(* IEC 61131-3 sources: cc_kush_rewrite/POUs (part 2) *)

// DO MODULES MAPPING (350-399)

// Модуль DO1 (350-351): Бункеры 1-2 - Управление ЧРП
FC_ModbusWriteBool(pRegisters := ADR(awModbusInputRegisters), iRegisterIndex := 350, iBitIndex := 0, xValue := stBunker[1].MotorVibFeeder[1].VFD.qxStart);
FC_ModbusWriteBool(pRegisters := ADR(awModbusInputRegisters), iRegisterIndex := 350, iBitIndex := 1, xValue := stBunker[1].MotorVibFeeder[1].VFD.qxResetFailure);
FC_ModbusWriteBool(pRegisters := ADR(awModbusInputRegisters), iRegisterIndex := 350, iBitIndex := 2, xValue := stBunker[1].MotorVibFeeder[2].VFD.qxStart);
FC_ModbusWriteBool(pRegisters := ADR(awModbusInputRegisters), iRegisterIndex := 350, iBitIndex := 3, xValue := stBunker[1].MotorVibFeeder[2].VFD.qxResetFailure);
FC_ModbusWriteBool(pRegisters := ADR(awModbusInputRegisters), iRegisterIndex := 350, iBitIndex := 4, xValue := stBunker[1].MotorVibrator[1].VFD.qxStart);
FC_ModbusWriteBool(pRegisters := ADR(awModbusInputRegisters), iRegisterIndex := 350, iBitIndex := 5, xValue := stBunker[1].MotorVibrator[1].VFD.qxResetFailure);
FC_ModbusWriteBool(pRegisters := ADR(awModbusInputRegisters), iRegisterIndex := 350, iBitIndex := 6, xValue := stBunker[1].MotorVibrator[2].VFD.qxStart);
FC_ModbusWriteBool(pRegisters := ADR(awModbusInputRegisters), iRegisterIndex := 350, iBitIndex := 7, xValue := stBunker[1].MotorVibrator[2].VFD.qxResetFailure);
FC_ModbusWriteBool(pRegisters := ADR(awModbusInputRegisters), iRegisterIndex := 350, iBitIndex := 8, xValue := stBunker[1].MotorVibrator[3].VFD.qxStart);
FC_ModbusWriteBool(pRegisters := ADR(awModbusInputRegisters), iRegisterIndex := 350, iBitIndex := 9, xValue := stBunker[1].MotorVibrator[3].VFD.qxResetFailure);
FC_ModbusWriteBool(pRegisters := ADR(awModbusInputRegisters), iRegisterIndex := 350, iBitIndex := 10, xValue := stBunker[1].MotorVibrator[4].VFD.qxStart);
FC_ModbusWriteBool(pRegisters := ADR(awModbusInputRegisters), iRegisterIndex := 350, iBitIndex := 11, xValue := stBunker[1].MotorVibrator[4].VFD.qxResetFailure);
FC_ModbusWriteBool(pRegisters := ADR(awModbusInputRegisters), iRegisterIndex := 350, iBitIndex := 12, xValue := stBunker[2].MotorVibFeeder[1].VFD.qxStart);
FC_ModbusWriteBool(pRegisters := ADR(awModbusInputRegisters), iRegisterIndex := 350, iBitIndex := 13, xValue := stBunker[2].MotorVibFeeder[1].VFD.qxResetFailure);
FC_ModbusWriteBool(pRegisters := ADR(awModbusInputRegisters), iRegisterIndex := 350, iBitIndex := 14, xValue := stBunker[2].MotorVibFeeder[2].VFD.qxStart);
FC_ModbusWriteBool(pRegisters := ADR(awModbusInputRegisters), iRegisterIndex := 350, iBitIndex := 15, xValue := stBunker[2].MotorVibFeeder[2].VFD.qxResetFailure);

FC_ModbusWriteBool(pRegisters := ADR(awModbusInputRegisters), iRegisterIndex := 351, iBitIndex := 0, xValue := stBunker[2].MotorVibrator[1].VFD.qxStart);
FC_ModbusWriteBool(pRegisters := ADR(awModbusInputRegisters), iRegisterIndex := 351, iBitIndex := 1, xValue := stBunker[2].MotorVibrator[1].VFD.qxResetFailure);
FC_ModbusWriteBool(pRegisters := ADR(awModbusInputRegisters), iRegisterIndex := 351, iBitIndex := 2, xValue := stBunker[2].MotorVibrator[2].VFD.qxStart);
FC_ModbusWriteBool(pRegisters := ADR(awModbusInputRegisters), iRegisterIndex := 351, iBitIndex := 3, xValue := stBunker[2].MotorVibrator[2].VFD.qxResetFailure);
FC_ModbusWriteBool(pRegisters := ADR(awModbusInputRegisters), iRegisterIndex := 351, iBitIndex := 4, xValue := stBunker[2].MotorVibrator[3].VFD.qxStart);
FC_ModbusWriteBool(pRegisters := ADR(awModbusInputRegisters), iRegisterIndex := 351, iBitIndex := 5, xValue := stBunker[2].MotorVibrator[3].VFD.qxResetFailure);
FC_ModbusWriteBool(pRegisters := ADR(awModbusInputRegisters), iRegisterIndex := 351, iBitIndex := 6, xValue := stBunker[2].MotorVibrator[4].VFD.qxStart);
FC_ModbusWriteBool(pRegisters := ADR(awModbusInputRegisters), iRegisterIndex := 351, iBitIndex := 7, xValue := stBunker[2].MotorVibrator[4].VFD.qxResetFailure);

// Модуль DO2 (352-353): Бункер 3, Конвейер, Отвалообразователь - Управление ЧРП
FC_ModbusWriteBool(pRegisters := ADR(awModbusInputRegisters), iRegisterIndex := 352, iBitIndex := 0, xValue := stBunker[3].MotorVibFeeder[1].VFD.qxStart);
FC_ModbusWriteBool(pRegisters := ADR(awModbusInputRegisters), iRegisterIndex := 352, iBitIndex := 1, xValue := stBunker[3].MotorVibFeeder[1].VFD.qxResetFailure);
FC_ModbusWriteBool(pRegisters := ADR(awModbusInputRegisters), iRegisterIndex := 352, iBitIndex := 2, xValue := stBunker[3].MotorVibFeeder[2].VFD.qxStart);
FC_ModbusWriteBool(pRegisters := ADR(awModbusInputRegisters), iRegisterIndex := 352, iBitIndex := 3, xValue := stBunker[3].MotorVibFeeder[2].VFD.qxResetFailure);
FC_ModbusWriteBool(pRegisters := ADR(awModbusInputRegisters), iRegisterIndex := 352, iBitIndex := 4, xValue := stBunker[3].MotorVibrator[1].VFD.qxStart);
FC_ModbusWriteBool(pRegisters := ADR(awModbusInputRegisters), iRegisterIndex := 352, iBitIndex := 5, xValue := stBunker[3].MotorVibrator[1].VFD.qxResetFailure);
FC_ModbusWriteBool(pRegisters := ADR(awModbusInputRegisters), iRegisterIndex := 352, iBitIndex := 6, xValue := stBunker[3].MotorVibrator[2].VFD.qxStart);
FC_ModbusWriteBool(pRegisters := ADR(awModbusInputRegisters), iRegisterIndex := 352, iBitIndex := 7, xValue := stBunker[3].MotorVibrator[2].VFD.qxResetFailure);
FC_ModbusWriteBool(pRegisters := ADR(awModbusInputRegisters), iRegisterIndex := 352, iBitIndex := 8, xValue := stBunker[3].MotorVibrator[3].VFD.qxStart);
FC_ModbusWriteBool(pRegisters := ADR(awModbusInputRegisters), iRegisterIndex := 352, iBitIndex := 9, xValue := stBunker[3].MotorVibrator[3].VFD.qxResetFailure);
FC_ModbusWriteBool(pRegisters := ADR(awModbusInputRegisters), iRegisterIndex := 352, iBitIndex := 10, xValue := stBunker[3].MotorVibrator[4].VFD.qxStart);
FC_ModbusWriteBool(pRegisters := ADR(awModbusInputRegisters), iRegisterIndex := 352, iBitIndex := 11, xValue := stBunker[3].MotorVibrator[4].VFD.qxResetFailure);
FC_ModbusWriteBool(pRegisters := ADR(awModbusInputRegisters), iRegisterIndex := 352, iBitIndex := 12, xValue := stConveyor.MotorConveyor[1].VFD.qxStart);
FC_ModbusWriteBool(pRegisters := ADR(awModbusInputRegisters), iRegisterIndex := 352, iBitIndex := 13, xValue := stConveyor.MotorConveyor[1].VFD.qxResetFailure);
FC_ModbusWriteBool(pRegisters := ADR(awModbusInputRegisters), iRegisterIndex := 352, iBitIndex := 14, xValue := stConveyor.MotorConveyor[2].VFD.qxStart);
FC_ModbusWriteBool(pRegisters := ADR(awModbusInputRegisters), iRegisterIndex := 352, iBitIndex := 15, xValue := stConveyor.MotorConveyor[2].VFD.qxResetFailure);

FC_ModbusWriteBool(pRegisters := ADR(awModbusInputRegisters), iRegisterIndex := 353, iBitIndex := 0, xValue := stDumper.MotorConveyor[1].VFD.qxStart);
FC_ModbusWriteBool(pRegisters := ADR(awModbusInputRegisters), iRegisterIndex := 353, iBitIndex := 1, xValue := stDumper.MotorConveyor[1].VFD.qxResetFailure);
FC_ModbusWriteBool(pRegisters := ADR(awModbusInputRegisters), iRegisterIndex := 353, iBitIndex := 2, xValue := stDumper.MotorConveyor[2].VFD.qxStart);
FC_ModbusWriteBool(pRegisters := ADR(awModbusInputRegisters), iRegisterIndex := 353, iBitIndex := 3, xValue := stDumper.MotorConveyor[2].VFD.qxResetFailure);
FC_ModbusWriteBool(pRegisters := ADR(awModbusInputRegisters), iRegisterIndex := 353, iBitIndex := 4, xValue := stDumper.MotorRotation[1].VFD.qxStart);
FC_ModbusWriteBool(pRegisters := ADR(awModbusInputRegisters), iRegisterIndex := 353, iBitIndex := 5, xValue := stDumper.MotorRotation[1].qxVFDReverseStart);
FC_ModbusWriteBool(pRegisters := ADR(awModbusInputRegisters), iRegisterIndex := 353, iBitIndex := 6, xValue := stDumper.MotorRotation[1].VFD.qxResetFailure);
FC_ModbusWriteBool(pRegisters := ADR(awModbusInputRegisters), iRegisterIndex := 353, iBitIndex := 7, xValue := stDumper.MotorRotation[2].VFD.qxStart);
FC_ModbusWriteBool(pRegisters := ADR(awModbusInputRegisters), iRegisterIndex := 353, iBitIndex := 8, xValue := stDumper.MotorRotation[2].qxVFDReverseStart);
FC_ModbusWriteBool(pRegisters := ADR(awModbusInputRegisters), iRegisterIndex := 353, iBitIndex := 9, xValue := stDumper.MotorRotation[2].VFD.qxResetFailure);

// Модуль DO3 (354-355): Контакторы и общие выходы
FC_ModbusWriteBool(pRegisters := ADR(awModbusInputRegisters), iRegisterIndex := 354, iBitIndex := 0, xValue := stConveyor.MotorConveyor[1].qxKM_Power);
FC_ModbusWriteBool(pRegisters := ADR(awModbusInputRegisters), iRegisterIndex := 354, iBitIndex := 1, xValue := stConveyor.MotorConveyor[2].qxKM_Power);
FC_ModbusWriteBool(pRegisters := ADR(awModbusInputRegisters), iRegisterIndex := 354, iBitIndex := 2, xValue := stDumper.MotorConveyor[1].qxKM_Power);
FC_ModbusWriteBool(pRegisters := ADR(awModbusInputRegisters), iRegisterIndex := 354, iBitIndex := 3, xValue := stDumper.MotorConveyor[2].qxKM_Power);
FC_ModbusWriteBool(pRegisters := ADR(awModbusInputRegisters), iRegisterIndex := 354, iBitIndex := 4, xValue := stDumper.MotorRotation[1].qxKM_Power);
FC_ModbusWriteBool(pRegisters := ADR(awModbusInputRegisters), iRegisterIndex := 354, iBitIndex := 5, xValue := stDumper.MotorRotation[2].qxKM_Power);
FC_ModbusWriteBool(pRegisters := ADR(awModbusInputRegisters), iRegisterIndex := 354, iBitIndex := 6, xValue := stBunker[1].MotorVibFeeder[1].qxKM_Power);
FC_ModbusWriteBool(pRegisters := ADR(awModbusInputRegisters), iRegisterIndex := 354, iBitIndex := 7, xValue := stBunker[1].MotorVibFeeder[2].qxKM_Power);
FC_ModbusWriteBool(pRegisters := ADR(awModbusInputRegisters), iRegisterIndex := 354, iBitIndex := 8, xValue := stBunker[1].MotorVibrator[1].qxKM_Power);
FC_ModbusWriteBool(pRegisters := ADR(awModbusInputRegisters), iRegisterIndex := 354, iBitIndex := 9, xValue := stBunker[1].MotorVibrator[2].qxKM_Power);
FC_ModbusWriteBool(pRegisters := ADR(awModbusInputRegisters), iRegisterIndex := 354, iBitIndex := 10, xValue := stBunker[1].MotorVibrator[3].qxKM_Power);
FC_ModbusWriteBool(pRegisters := ADR(awModbusInputRegisters), iRegisterIndex := 354, iBitIndex := 11, xValue := stBunker[1].MotorVibrator[4].qxKM_Power);
FC_ModbusWriteBool(pRegisters := ADR(awModbusInputRegisters), iRegisterIndex := 354, iBitIndex := 12, xValue := stBunker[2].MotorVibFeeder[1].qxKM_Power);
FC_ModbusWriteBool(pRegisters := ADR(awModbusInputRegisters), iRegisterIndex := 354, iBitIndex := 13, xValue := stBunker[2].MotorVibFeeder[2].qxKM_Power);
FC_ModbusWriteBool(pRegisters := ADR(awModbusInputRegisters), iRegisterIndex := 354, iBitIndex := 14, xValue := stBunker[2].MotorVibrator[1].qxKM_Power);
FC_ModbusWriteBool(pRegisters := ADR(awModbusInputRegisters), iRegisterIndex := 354, iBitIndex := 15, xValue := stBunker[2].MotorVibrator[2].qxKM_Power);

FC_ModbusWriteBool(pRegisters := ADR(awModbusInputRegisters), iRegisterIndex := 355, iBitIndex := 0, xValue := stBunker[2].MotorVibrator[3].qxKM_Power);
FC_ModbusWriteBool(pRegisters := ADR(awModbusInputRegisters), iRegisterIndex := 355, iBitIndex := 1, xValue := stBunker[2].MotorVibrator[4].qxKM_Power);
FC_ModbusWriteBool(pRegisters := ADR(awModbusInputRegisters), iRegisterIndex := 355, iBitIndex := 2, xValue := stBunker[3].MotorVibFeeder[1].qxKM_Power);
FC_ModbusWriteBool(pRegisters := ADR(awModbusInputRegisters), iRegisterIndex := 355, iBitIndex := 3, xValue := stBunker[3].MotorVibFeeder[2].qxKM_Power);
FC_ModbusWriteBool(pRegisters := ADR(awModbusInputRegisters), iRegisterIndex := 355, iBitIndex := 4, xValue := stBunker[3].MotorVibrator[1].qxKM_Power);
FC_ModbusWriteBool(pRegisters := ADR(awModbusInputRegisters), iRegisterIndex := 355, iBitIndex := 5, xValue := stBunker[3].MotorVibrator[2].qxKM_Power);
FC_ModbusWriteBool(pRegisters := ADR(awModbusInputRegisters), iRegisterIndex := 355, iBitIndex := 6, xValue := stBunker[3].MotorVibrator[3].qxKM_Power);
FC_ModbusWriteBool(pRegisters := ADR(awModbusInputRegisters), iRegisterIndex := 355, iBitIndex := 7, xValue := stBunker[3].MotorVibrator[4].qxKM_Power);
FC_ModbusWriteBool(pRegisters := ADR(awModbusInputRegisters), iRegisterIndex := 355, iBitIndex := 8, xValue := stConveyor.xHLA);
FC_ModbusWriteBool(pRegisters := ADR(awModbusInputRegisters), iRegisterIndex := 355, iBitIndex := 10, xValue := stDumper.xHLA);
FC_ModbusWriteBool(pRegisters := ADR(awModbusInputRegisters), iRegisterIndex := 355, iBitIndex := 11, xValue := stCommonSignals.qx6KM1);
FC_ModbusWriteBool(pRegisters := ADR(awModbusInputRegisters), iRegisterIndex := 355, iBitIndex := 12, xValue := stConveyor.qxBreakerConveyor);
FC_ModbusWriteBool(pRegisters := ADR(awModbusInputRegisters), iRegisterIndex := 355, iBitIndex := 13, xValue := stDumper.qxBreakerConveyor);
FC_ModbusWriteBool(pRegisters := ADR(awModbusInputRegisters), iRegisterIndex := 355, iBitIndex := 14, xValue := stDumper.qxBreakerRotation);

// Модуль DO4 (356-357): Светофоры бункеров
FC_ModbusWriteBool(pRegisters := ADR(awModbusInputRegisters), iRegisterIndex := 356, iBitIndex := 0, xValue := stBunker[1].qxLightRed);
FC_ModbusWriteBool(pRegisters := ADR(awModbusInputRegisters), iRegisterIndex := 356, iBitIndex := 1, xValue := stBunker[1].qxLightYellow);
FC_ModbusWriteBool(pRegisters := ADR(awModbusInputRegisters), iRegisterIndex := 356, iBitIndex := 2, xValue := stBunker[1].qxLightGreen);
FC_ModbusWriteBool(pRegisters := ADR(awModbusInputRegisters), iRegisterIndex := 356, iBitIndex := 3, xValue := stBunker[2].qxLightRed);
FC_ModbusWriteBool(pRegisters := ADR(awModbusInputRegisters), iRegisterIndex := 356, iBitIndex := 4, xValue := stBunker[2].qxLightYellow);
FC_ModbusWriteBool(pRegisters := ADR(awModbusInputRegisters), iRegisterIndex := 356, iBitIndex := 5, xValue := stBunker[2].qxLightGreen);
FC_ModbusWriteBool(pRegisters := ADR(awModbusInputRegisters), iRegisterIndex := 356, iBitIndex := 6, xValue := stBunker[3].qxLightRed);
FC_ModbusWriteBool(pRegisters := ADR(awModbusInputRegisters), iRegisterIndex := 356, iBitIndex := 7, xValue := stBunker[3].qxLightYellow);
FC_ModbusWriteBool(pRegisters := ADR(awModbusInputRegisters), iRegisterIndex := 356, iBitIndex := 8, xValue := stBunker[3].qxLightGreen);

END_FUNCTION

(* ---- FB_BunkerControl.st ---- *)
FUNCTION_BLOCK FB_BunkerControl
VAR_INPUT
	Bunker : REFERENCE TO ST_Bunker;
	xLocalMode : BOOL; // TRUE = местный режим (ПМУ), FALSE = дистанционный режим (SCADA)
	xStart : BOOL; // Команда запуска вибропитателей (дистанционный режим)
	xStop : BOOL; // Команда остановки (дистанционный режим)
	xEmergencyStopVibFeeder : BOOL; // Аварийная остановка вибропитателей (переводит бункер в ERROR)
	xEmergencyStopVibrator : BOOL; // Аварийная остановка вибраторов (только отключает вибраторы)
	xReset : BOOL; // Сброс ошибок
	irManualFrequency : REAL; // Частота вибропитателей для ручного режима управления
	irManualFrequencyVibrator : REAL; // Частота вибраторов для ручного режима управления
END_VAR
VAR_OUTPUT
	eStage : E_StageWithPreStartAlarm; // Текущая стадия запуска вибропитателей
	eStageToSCADA : E_ScadaStatesDevice; // Передача состояния скаде
END_VAR
VAR
	i : INT;
	_rtStartCmd, _rtStopCmd : R_TRIG; // Детекторы фронтов для команд

	// Локальные переменные для управления в режиме МЕСТНЫЙ
	_rtStartKM, _rtStopKM : R_TRIG;
	_rtStartVFD, _rtStopVFD : R_TRIG;

	// Объединенные команды (ПМУ или SCADA в зависимости от режима)
	xStartCommand : BOOL; // Фактическая команда запуска (из ПМУ или SCADA)
	xStopCommand : BOOL; // Фактическая команда остановки (из ПМУ или SCADA)

	// ФБ управления
	fbPneumoControl : FB_PneumoCollapseControl;

	// Таймеры для автоматического цикла вибраторов
	tonVibratorActive : TON;  // Таймер активной работы вибраторов
	tonVibratorPause : TON;   // Таймер паузы вибраторов

	// Автомат состояний для запуска вибропитателей
	STAGE : E_StageWithPreStartAlarm := E_StageWithPreStartAlarm.IDLE;

	// Состояние схемы контакторов (TRUE = схема собрана, FALSE = схема разобрана)
	xCircuitBuilt : BOOL := FALSE;
	xCircuitBuiltVibrator : BOOL := FALSE;

	// Целевые частоты для моторов вибропитателей
	rTargetFreqVibFeeder1 : REAL := 0.0;
	rTargetFreqVibFeeder2 : REAL := 0.0;

	// Флаг активного запуска вибраторов в ручном режиме
	xVibratorManualRunActive : BOOL := FALSE;

	// Флаг текущей активности вибраторов в автоматическом режиме
	xVibratorAutoActive : BOOL := FALSE;

	// Таймеры контроля выполнения команд
	fbTimerStarting : TON; // Тайм-аут запуска (STARTING → WORK)
	fbTimerStopping : TON; // Тайм-аут остановки (WORK → IDLE)

END_VAR

// ========================================
// FB_BunkerControl - Управление бункером
// ========================================
//
// РЕЖИМЫ УПРАВЛЕНИЯ:
//
// 1. МЕСТНЫЙ РЕЖИМ (xLocalMode = TRUE):
//    - Команды берутся с кнопок ПМУ (Bunker.fbBtnStart, fbBtnStop)
//    - ПУСК/СТОП вибропитателей по фронтам кнопок
//    - Автоматически устанавливает eStateRemote = Manual
//
// 2. ДИСТАНЦИОННЫЙ РЕЖИМ (xLocalMode = FALSE):
//    - Команды берутся из входов ФБ (xStart, xStop)
//    - Режим устанавливается через SCADA (Manual/Remote/Auto)
//
// УПРАВЛЕНИЕ ВИБРОПИТАТЕЛЯМИ:
// - ПУСК: включение вибропитателей с заданной частотой
// - СТОП: остановка вибропитателей
// - Частота: Auto - от ПИД, Manual/Repair - от irManualFrequency
//
// УПРАВЛЕНИЕ ВИБРАТОРАМИ:
// - Независимо от режима вибропитателей
// - Режимы:
//   * Auto - циклическая работа по таймеру (ACTIVE ↔ PAUSE)
//     - Работает только в стадии WORK вибропитателей
//     - Параметры: VIBRATOR_SETTINGS.TIME_ACTIVE, TIME_PAUSE_VIBRATOR
//     - Частота: irManualFrequencyVibrator
//   * Manual - выборочное управление через cmdAddVib1..4
//     - СТАРТ/СТОП по командам cmdStartVibrator/cmdStopVibrator
//     - Частота: irManualFrequencyVibrator
//   * Repair - все вибраторы остановлены
//
// ========================================

// ========================================
// ИНИЦИАЛИЗАЦИЯ СИГНАЛОВ С ФИЛЬТРАЦИЕЙ ДРЕБЕЗГА
// ========================================

// Положение люка - с фильтрацией дребезга
Bunker.fbStateHatch(
	ixSignal := , // Подключить физический вход
	xEnableRattlingFilter := TRUE,
	tStabilityTime := T#100MS
);

// ПМУ - СТАРТ - с фильтрацией дребезга
Bunker.fbBtnStart(
	ixSignal := , // Подключить физический вход
	xEnableRattlingFilter := TRUE,
	tStabilityTime := T#100MS
);

// ПМУ - СТОП - с фильтрацией дребезга
Bunker.fbBtnStop(
	ixSignal := , // Подключить физический вход
	xEnableRattlingFilter := TRUE,
	tStabilityTime := T#100MS
);

// ПМУ - Аварийная остановка - с фильтрацией дребезга
Bunker.fbBtnEmergencyStop(
	ixSignal := , // Подключить физический вход
	xEnableRattlingFilter := TRUE,
	tStabilityTime := T#100MS
);

// Двигатели вибраторов
FOR i := 1 TO AMOUNT_BUNKER_MOTOR_VIBRATOR BY 1 DO
	Bunker.MotorVibrator[i].fbStateKM(
		ixSignal := , // Состояние контактора
		xEnableRattlingFilter := TRUE
	);

	Bunker.MotorVibrator[i].fbStateQF(
		ixSignal := , // Автомат. выключатель
		xEnableRattlingFilter := TRUE
	);

	Bunker.MotorVibrator[i].VFD.fbStateFailure(
		ixSignal := , // ЧРП - ошибка
		xEnableRattlingFilter := TRUE
	);

	Bunker.MotorVibrator[i].VFD.fbStateRdyToStart(
		ixSignal := , // ЧРП - Готовность
		xEnableRattlingFilter := TRUE
	);

	Bunker.MotorVibrator[i].VFD.fbStateIsWorking(
		ixSignal := , // ЧРП - Работа
		xEnableRattlingFilter := TRUE
	);
END_FOR;

// Двигатели вибропитателей
FOR i := 1 TO AMOUNT_BUNKER_MOTOR_VIBFEEDER BY 1 DO
	Bunker.MotorVibFeeder[i].fbStateKM(
		ixSignal := , // Состояние контактора
		xEnableRattlingFilter := TRUE
	);

	Bunker.MotorVibFeeder[i].fbStatorOverheat(
		ixSignal := , // Перегрев статора
		xEnableRattlingFilter := TRUE
	);

	Bunker.MotorVibFeeder[i].fbStateQF(
		ixSignal := , // Автомат. выключатель
		xEnableRattlingFilter := TRUE
	);

	Bunker.MotorVibFeeder[i].VFD.fbStateFailure(
		ixSignal := , // ЧРП - ошибка
		xEnableRattlingFilter := TRUE
	);

	Bunker.MotorVibFeeder[i].VFD.fbStateRdyToStart(
		ixSignal := , // ЧРП - Готовность
		xEnableRattlingFilter := TRUE
	);

	Bunker.MotorVibFeeder[i].VFD.fbStateIsWorking(
		ixSignal := , // ЧРП - Работа
		xEnableRattlingFilter := TRUE
	);

	// Device control для контакторов
	Bunker.MotorVibFeeder[i].Device(
		ixFeedback := Bunker.MotorVibFeeder[i].fbStateKM.qxSignal,
		xEnableFeedback := TRUE
	);
END_FOR;

// ========================================
// ОБРАБОТКА ДИАГНОСТИКИ ДИАПАЗОНОВ
// ========================================

// Аналоговые входы температуры подшипникового узла мотора вибропитателя 1
Bunker.MotorVibFeeder[1].fbAnalogInput[1](
	xSimulation := SIMULATION,
	iADC_Code := Bunker.MotorVibFeeder[1].nTempBearingRawSignal[1],
	refEngValue := Bunker.MotorVibFeeder[1].rTempBearing[1],
	refSimValue := Bunker.MotorVibFeeder[1].rSimulatedTempBearing[1],
	rAlarm_LL := VFD_CURRENT_ALARM_LL,
	rAlarm_L := VFD_CURRENT_ALARM_L,
	rAlarm_H := VFD_CURRENT_ALARM_H,
	rAlarm_HH := VFD_CURRENT_ALARM_HH,
	iADC_Max := VFD_ADC_MAX,
	iADC_Min := VFD_ADC_MIN,
	rEngValue_Max := TEMP_BEARING_MAX,
	rEngValue_Min := TEMP_BEARING_MIN,
	rCurrent_Max := VFD_CURRENT_MAX,
	rCurrent_Min := VFD_CURRENT_MIN
);

Bunker.MotorVibFeeder[1].fbAnalogInput[2](
	xSimulation := SIMULATION,
	iADC_Code := Bunker.MotorVibFeeder[1].nTempBearingRawSignal[2],
	refEngValue := Bunker.MotorVibFeeder[1].rTempBearing[2],
	refSimValue := Bunker.MotorVibFeeder[1].rSimulatedTempBearing[2],
	rAlarm_LL := VFD_CURRENT_ALARM_LL,
	rAlarm_L := VFD_CURRENT_ALARM_L,
	rAlarm_H := VFD_CURRENT_ALARM_H,
	rAlarm_HH := VFD_CURRENT_ALARM_HH,
	iADC_Max := VFD_ADC_MAX,
	iADC_Min := VFD_ADC_MIN,
	rEngValue_Max := TEMP_BEARING_MAX,
	rEngValue_Min := TEMP_BEARING_MIN,
	rCurrent_Max := VFD_CURRENT_MAX,
	rCurrent_Min := VFD_CURRENT_MIN
);

// Проверки LL HH мотора вибропитателя 1
Bunker.MotorVibFeeder[1].fbRangeDiagnostic[1](
	irValue := Bunker.MotorVibFeeder[1].rTempBearing[1],
	irSetpointL := MOTOR_VIBFEEDER_TEMP_POINTS.L_Value,
	irSetpointLL := MOTOR_VIBFEEDER_TEMP_POINTS.LL_Value,
	irSetpointH := MOTOR_VIBFEEDER_TEMP_POINTS.H_Value,
	irSetpointHH := MOTOR_VIBFEEDER_TEMP_POINTS.HH_Value,
	ixEnable := TRUE
);

Bunker.MotorVibFeeder[1].fbRangeDiagnostic[2](
	irValue := Bunker.MotorVibFeeder[1].rTempBearing[2],
	irSetpointL := MOTOR_VIBFEEDER_TEMP_POINTS.L_Value,
	irSetpointLL := MOTOR_VIBFEEDER_TEMP_POINTS.LL_Value,
	irSetpointH := MOTOR_VIBFEEDER_TEMP_POINTS.H_Value,
	irSetpointHH := MOTOR_VIBFEEDER_TEMP_POINTS.HH_Value,
	ixEnable := TRUE
);

Bunker.MotorVibFeeder[1].VFD.fbRangeDiagnostic(
	irValue := Bunker.MotorVibFeeder[1].VFD.wMotorCurrent.rTag,
	irSetpointL := MOTOR_VIBFEEDER_CURRENT_POINTS.L_Value,
	irSetpointLL := MOTOR_VIBFEEDER_CURRENT_POINTS.LL_Value,
	irSetpointH := MOTOR_VIBFEEDER_CURRENT_POINTS.H_Value,
	irSetpointHH := MOTOR_VIBFEEDER_CURRENT_POINTS.HH_Value,
	ixEnable := TRUE
);

// Аналоговый вход ЧРП (чтение текущей частоты)
Bunker.MotorVibFeeder[1].VFD.fbAnalogInput(
	xSimulation := SIMULATION,
	iADC_Code := Bunker.MotorVibFeeder[1].VFD.nActualFrequencyADC,
	refEngValue := Bunker.MotorVibFeeder[1].VFD.rActualFrequency,
	refSimValue := Bunker.MotorVibFeeder[1].VFD.rSimulatedFrequency,
	rAlarm_LL := VFD_CURRENT_ALARM_LL,
	rAlarm_L := VFD_CURRENT_ALARM_L,
	rAlarm_H := VFD_CURRENT_ALARM_H,
	rAlarm_HH := VFD_CURRENT_ALARM_HH,
	iADC_Max := VFD_ADC_MAX,
	iADC_Min := VFD_ADC_MIN,
	rEngValue_Max := VFD_FREQ_MAX_RANGE,
	rEngValue_Min := VFD_FREQ_MIN,
	rCurrent_Max := VFD_CURRENT_MAX,
	rCurrent_Min := VFD_CURRENT_MIN
);

// Аналоговый выход ЧРП (задание частоты)
Bunker.MotorVibFeeder[1].VFD.fbAnalogOutput(
	xEnable := Bunker.MotorVibFeeder[1].VFD.fbStateIsWorking.qxSignal,
	rEngValue := Bunker.MotorVibFeeder[1].VFD.Frequency.qrCurrentFrequency,
	rEngValue_Max := VFD_FREQ_MAX_RANGE,
	rEngValue_Min := VFD_FREQ_MIN,
	rCurrent_Max := VFD_CURRENT_MAX,
	rCurrent_Min := VFD_CURRENT_MIN,
	iDAC_Max := VFD_ADC_MAX,
	iDAC_Min := VFD_ADC_MIN,
	rAlarm_LL := VFD_CURRENT_ALARM_LL,
	rAlarm_L := VFD_CURRENT_ALARM_L,
	rAlarm_H := VFD_CURRENT_ALARM_H,
	rAlarm_HH := VFD_CURRENT_ALARM_HH,
	xEnableClamp := TRUE
);
Bunker.MotorVibFeeder[1].VFD.nSetOutSignalToModule := Bunker.MotorVibFeeder[1].VFD.fbAnalogOutput.iDAC_Code;

// Аналоговые входы температуры подшипникового узла мотора вибропитателя 2
Bunker.MotorVibFeeder[2].fbAnalogInput[1](
	xSimulation := SIMULATION,
	iADC_Code := Bunker.MotorVibFeeder[2].nTempBearingRawSignal[1],
	refEngValue := Bunker.MotorVibFeeder[2].rTempBearing[1],
	refSimValue := Bunker.MotorVibFeeder[2].rSimulatedTempBearing[1],
	rAlarm_LL := VFD_CURRENT_ALARM_LL,
	rAlarm_L := VFD_CURRENT_ALARM_L,
	rAlarm_H := VFD_CURRENT_ALARM_H,
	rAlarm_HH := VFD_CURRENT_ALARM_HH,
	iADC_Max := VFD_ADC_MAX,
	iADC_Min := VFD_ADC_MIN,
	rEngValue_Max := TEMP_BEARING_MAX,
	rEngValue_Min := TEMP_BEARING_MIN,
	rCurrent_Max := VFD_CURRENT_MAX,
	rCurrent_Min := VFD_CURRENT_MIN
);

Bunker.MotorVibFeeder[2].fbAnalogInput[2](
	xSimulation := SIMULATION,
	iADC_Code := Bunker.MotorVibFeeder[2].nTempBearingRawSignal[2],
	refEngValue := Bunker.MotorVibFeeder[2].rTempBearing[2],
	refSimValue := Bunker.MotorVibFeeder[2].rSimulatedTempBearing[2],
	rAlarm_LL := VFD_CURRENT_ALARM_LL,
	rAlarm_L := VFD_CURRENT_ALARM_L,
	rAlarm_H := VFD_CURRENT_ALARM_H,
	rAlarm_HH := VFD_CURRENT_ALARM_HH,
	iADC_Max := VFD_ADC_MAX,
	iADC_Min := VFD_ADC_MIN,
	rEngValue_Max := TEMP_BEARING_MAX,
	rEngValue_Min := TEMP_BEARING_MIN,
	rCurrent_Max := VFD_CURRENT_MAX,
	rCurrent_Min := VFD_CURRENT_MIN
);

// Проверки LL HH мотора вибропитателя 2
Bunker.MotorVibFeeder[2].fbRangeDiagnostic[1](
	irValue := Bunker.MotorVibFeeder[2].rTempBearing[1],
	irSetpointL := MOTOR_VIBFEEDER_TEMP_POINTS.L_Value,
	irSetpointLL := MOTOR_VIBFEEDER_TEMP_POINTS.LL_Value,
	irSetpointH := MOTOR_VIBFEEDER_TEMP_POINTS.H_Value,
	irSetpointHH := MOTOR_VIBFEEDER_TEMP_POINTS.HH_Value,
	ixEnable := TRUE
);

Bunker.MotorVibFeeder[2].fbRangeDiagnostic[2](
	irValue := Bunker.MotorVibFeeder[2].rTempBearing[2],
	irSetpointL := MOTOR_VIBFEEDER_TEMP_POINTS.L_Value,
	irSetpointLL := MOTOR_VIBFEEDER_TEMP_POINTS.LL_Value,
	irSetpointH := MOTOR_VIBFEEDER_TEMP_POINTS.H_Value,
	irSetpointHH := MOTOR_VIBFEEDER_TEMP_POINTS.HH_Value,
	ixEnable := TRUE
);

Bunker.MotorVibFeeder[2].VFD.fbRangeDiagnostic(
	irValue := Bunker.MotorVibFeeder[2].VFD.wMotorCurrent.rTag,
	irSetpointL := MOTOR_VIBFEEDER_CURRENT_POINTS.L_Value,
	irSetpointLL := MOTOR_VIBFEEDER_CURRENT_POINTS.LL_Value,
	irSetpointH := MOTOR_VIBFEEDER_CURRENT_POINTS.H_Value,
	irSetpointHH := MOTOR_VIBFEEDER_CURRENT_POINTS.HH_Value,
	ixEnable := TRUE
);

// Аналоговый вход ЧРП (чтение текущей частоты)
Bunker.MotorVibFeeder[2].VFD.fbAnalogInput(
	xSimulation := SIMULATION,
	iADC_Code := Bunker.MotorVibFeeder[2].VFD.nActualFrequencyADC,
	refEngValue := Bunker.MotorVibFeeder[2].VFD.rActualFrequency,
	refSimValue := Bunker.MotorVibFeeder[2].VFD.rSimulatedFrequency,
	rAlarm_LL := VFD_CURRENT_ALARM_LL,
	rAlarm_L := VFD_CURRENT_ALARM_L,
	rAlarm_H := VFD_CURRENT_ALARM_H,
	rAlarm_HH := VFD_CURRENT_ALARM_HH,
	iADC_Max := VFD_ADC_MAX,
	iADC_Min := VFD_ADC_MIN,
	rEngValue_Max := VFD_FREQ_MAX_RANGE,
	rEngValue_Min := VFD_FREQ_MIN,
	rCurrent_Max := VFD_CURRENT_MAX,
	rCurrent_Min := VFD_CURRENT_MIN
);

// Аналоговый выход ЧРП (задание частоты)
Bunker.MotorVibFeeder[2].VFD.fbAnalogOutput(
	xEnable := Bunker.MotorVibFeeder[2].VFD.fbStateIsWorking.qxSignal,
	rEngValue := Bunker.MotorVibFeeder[2].VFD.Frequency.qrCurrentFrequency,
	rEngValue_Max := VFD_FREQ_MAX_RANGE,
	rEngValue_Min := VFD_FREQ_MIN,
	rCurrent_Max := VFD_CURRENT_MAX,
	rCurrent_Min := VFD_CURRENT_MIN,
	iDAC_Max := VFD_ADC_MAX,
	iDAC_Min := VFD_ADC_MIN,
	rAlarm_LL := VFD_CURRENT_ALARM_LL,
	rAlarm_L := VFD_CURRENT_ALARM_L,
	rAlarm_H := VFD_CURRENT_ALARM_H,
	rAlarm_HH := VFD_CURRENT_ALARM_HH,
	xEnableClamp := TRUE
);
Bunker.MotorVibFeeder[2].VFD.nSetOutSignalToModule := Bunker.MotorVibFeeder[2].VFD.fbAnalogOutput.iDAC_Code;

// Проверки LL HH моторов вибратора
FOR i := 1 TO AMOUNT_BUNKER_MOTOR_VIBRATOR BY 1 DO
	Bunker.MotorVibrator[i].VFD.fbRangeDiagnostic(
		irValue := Bunker.MotorVibrator[i].VFD.wMotorCurrent.rTag,
		irSetpointL := MOTOR_VIBRATOR_CURRENT_POINTS.L_Value,
		irSetpointLL := MOTOR_VIBRATOR_CURRENT_POINTS.LL_Value,
		irSetpointH := MOTOR_VIBRATOR_CURRENT_POINTS.H_Value,
		irSetpointHH := MOTOR_VIBRATOR_CURRENT_POINTS.HH_Value,
		ixEnable := TRUE
	);

	// Аналоговый вход ЧРП (чтение текущей частоты)
	Bunker.MotorVibrator[i].VFD.fbAnalogInput(
		xSimulation := SIMULATION,
		iADC_Code := Bunker.MotorVibrator[i].VFD.nActualFrequencyADC,
		refEngValue := Bunker.MotorVibrator[i].VFD.rActualFrequency,
		refSimValue := Bunker.MotorVibrator[i].VFD.rSimulatedFrequency,
		rAlarm_LL := VFD_CURRENT_ALARM_LL,
		rAlarm_L := VFD_CURRENT_ALARM_L,
		rAlarm_H := VFD_CURRENT_ALARM_H,
		rAlarm_HH := VFD_CURRENT_ALARM_HH,
		iADC_Max := VFD_ADC_MAX,
		iADC_Min := VFD_ADC_MIN,
		rEngValue_Max := VFD_FREQ_MAX_RANGE,
		rEngValue_Min := VFD_FREQ_MIN,
		rCurrent_Max := VFD_CURRENT_MAX,
		rCurrent_Min := VFD_CURRENT_MIN
	);

	// Аналоговый выход ЧРП (задание частоты)
	Bunker.MotorVibrator[i].VFD.fbAnalogOutput(
		xEnable := Bunker.MotorVibrator[i].VFD.fbStateIsWorking.qxSignal,
		rEngValue := Bunker.MotorVibrator[i].VFD.qrOutFrequency,
		rEngValue_Max := VFD_FREQ_MAX_RANGE,
		rEngValue_Min := VFD_FREQ_MIN,
		rCurrent_Max := VFD_CURRENT_MAX,
		rCurrent_Min := VFD_CURRENT_MIN,
		iDAC_Max := VFD_ADC_MAX,
		iDAC_Min := VFD_ADC_MIN,
		rAlarm_LL := VFD_CURRENT_ALARM_LL,
		rAlarm_L := VFD_CURRENT_ALARM_L,
		rAlarm_H := VFD_CURRENT_ALARM_H,
		rAlarm_HH := VFD_CURRENT_ALARM_HH,
		xEnableClamp := TRUE
	);
	Bunker.MotorVibrator[i].VFD.nSetOutSignalToModule := Bunker.MotorVibrator[i].VFD.fbAnalogOutput.iDAC_Code;
END_FOR;

fbPneumoControl(
	xEnable:= ,
	xManualStart:= ,
	tActiveTime:= VIBRATOR_SETTINGS.TIME_ACTIVE,
	tPauseCycle:= VIBRATOR_SETTINGS.TIME_PAUSE_VIBRATOR,
	tPauseFB:= VIBRATOR_SETTINGS.TIME_PAUSE_FB,
	nCycleCount:= VIBRATOR_SETTINGS.COUNT_CYCLE,
	xPneumoActive=> ,
	tTimeToNext=> );

// ========================================
// ОПРЕДЕЛЕНИЕ СОСТОЯНИЙ ДЛЯ SCADA
// ========================================

// Проверка ошибок вибропитателей (без вибраторов и пневмообрушения)
//	Bunker.xStateFailure := FC_Bunker_GetErrorMotorVibFeeder(Bunker := Bunker)
//					 OR FC_Bunker_GetErrorBunker(Bunker := Bunker);

// Проверка предупреждений вибропитателей:
// 1. Контроль тока моторов вибропитателей - уровень L или H
// 2. Температура подшипников - уровень L или H
Bunker.xStateWarning := Bunker.MotorVibFeeder[1].VFD.fbRangeDiagnostic.qxWarningActive
                     OR Bunker.MotorVibFeeder[2].VFD.fbRangeDiagnostic.qxWarningActive
                     OR Bunker.MotorVibFeeder[1].fbRangeDiagnostic[1].qxWarningActive
                     OR Bunker.MotorVibFeeder[1].fbRangeDiagnostic[2].qxWarningActive
                     OR Bunker.MotorVibFeeder[2].fbRangeDiagnostic[1].qxWarningActive
                     OR Bunker.MotorVibFeeder[2].fbRangeDiagnostic[2].qxWarningActive;

// ========================================
// ВЫБОР ИСТОЧНИКА КОМАНД (ПМУ ИЛИ SCADA)
// ========================================

// В местном режиме (xLocalMode = TRUE) - команды берутся с ПМУ (кнопки)
// В дистанционном режиме (xLocalMode = FALSE) - команды берутся из SCADA (входы ФБ)
IF xLocalMode THEN
	// Местный режим - команды с ПМУ
	xStartCommand := Bunker.fbBtnStart.qxRisingEdge; // ПУСК по фронту кнопки
	xStopCommand := Bunker.fbBtnStop.qxRisingEdge;   // СТОП по фронту кнопки
ELSE
	// Дистанционный режим - команды из SCADA
	xStartCommand := xStart;
	xStopCommand := xStop;
END_IF;

// ========================================
// АВТОМАТ СОСТОЯНИЙ ЗАПУСКА ВИБРОПИТАТЕЛЕЙ
// ========================================

// ПРИОРИТЕТНАЯ ПРОВЕРКА АВАРИЙНОЙ ОСТАНОВКИ ВИБРОПИТАТЕЛЕЙ
// Аварийная остановка питателей имеет наивысший приоритет и срабатывает в любой стадии
// 1. Внешний сигнал аварийной остановки (от SCADA или системы)
// 2. Кнопка аварийной остановки на ПМУ (NC контакт: FALSE = кнопка нажата)
//	IF xEmergencyStopVibFeeder OR NOT Bunker.fbBtnEmergencyStop.qxSignal THEN
//	STAGE := E_StageWithPreStartAlarm.ERROR;
//END_IF;

// ПРОВЕРКА ТАЙМ-АУТОВ ВЫПОЛНЕНИЯ КОМАНД
// Тайм-аут запуска: не удалось запустить вибропитатели за установленное время
IF fbTimerStarting.Q THEN
	STAGE := E_StageWithPreStartAlarm.ERROR;
END_IF;

// Тайм-аут остановки: не удалось остановить вибропитатели за установленное время
IF fbTimerStopping.Q THEN
	STAGE := E_StageWithPreStartAlarm.ERROR;
END_IF;

		// Обработка команды останова
		IF xStopCommand THEN
			// Запуск таймера остановки (тайм-аут на остановку вибропитателей)
			fbTimerStopping(
				IN := TRUE,
				PT := TIME_TIMEOUT_STOP_BUNKER
			);

			// Остановка VFD
			Bunker.MotorVibFeeder[1].VFD.qxStart := FALSE;
			Bunker.MotorVibFeeder[2].VFD.qxStart := FALSE;

			// Проверка остановки VFD (обратная связь)
			IF NOT Bunker.MotorVibFeeder[1].VFD.fbStateIsWorking.qxSignal
			   AND NOT Bunker.MotorVibFeeder[2].VFD.fbStateIsWorking.qxSignal
			THEN
				// Сброс таймера остановки (успешная остановка)
				fbTimerStopping(IN := FALSE);
				STAGE := E_StageWithPreStartAlarm.IDLE;
			END_IF;
		END_IF

CASE STAGE OF
	E_StageWithPreStartAlarm.IDLE:
		// Сброс таймеров запуска и остановки
		fbTimerStarting(IN := FALSE);
		fbTimerStopping(IN := FALSE);

		// Сброс целевых частот
		rTargetFreqVibFeeder1 := 0.0;
		rTargetFreqVibFeeder2 := 0.0;

		// Остановка VFD
		Bunker.MotorVibFeeder[1].VFD.qxStart := FALSE;
		Bunker.MotorVibFeeder[2].VFD.qxStart := FALSE;

		// Переход в STARTING при получении команды запуска
		IF xStartCommand THEN
			STAGE := E_StageWithPreStartAlarm.STARTING;
		END_IF

	E_StageWithPreStartAlarm.STARTING:
		// Запуск таймера запуска (тайм-аут на запуск вибропитателей)
		// Для бункеров используем соответствующую уставку (TIME_AFTER_START_BUNKER_1/2/3)
		// Но так как это общий FB, используем универсальную уставку
		fbTimerStarting(
			IN := TRUE,
			PT := TIME_AFTER_START_BUNKER_1 // Можно сделать параметром VAR_INPUT если нужно разные уставки для разных бункеров
		);

		// Команда ПУСК на VFD (TRUE = ПУСК)
		Bunker.MotorVibFeeder[1].VFD.qxStart := TRUE;
		Bunker.MotorVibFeeder[2].VFD.qxStart := TRUE;

		// Выбор источника частоты в зависимости от режима управления
		IF Bunker.eStateRemote = E_StateRemote.Auto THEN
			// Автоматический режим - частота от ПИД
			rTargetFreqVibFeeder1 := irManualFrequency; // TODO ВРЕМЕННО Bunker.rMotorVibFeederCommonFrequency
			rTargetFreqVibFeeder2 := irManualFrequency;
		ELSE
			// Ручной/Ремонт режим - частота от входного параметра irManualFrequency
			rTargetFreqVibFeeder1 := irManualFrequency;
			rTargetFreqVibFeeder2 := irManualFrequency;
		END_IF;

		// Переход в WORK по включению оборудования (обратная связь VFD)
		IF Bunker.MotorVibFeeder[1].VFD.fbStateIsWorking.qxSignal
		   AND Bunker.MotorVibFeeder[2].VFD.fbStateIsWorking.qxSignal
		THEN
			// Сброс таймера запуска (успешный запуск)
			fbTimerStarting(IN := FALSE);
			STAGE := E_StageWithPreStartAlarm.WORK;
		END_IF

	E_StageWithPreStartAlarm.WORK:

		// Выбор источника частоты в зависимости от режима управления
		IF Bunker.eStateRemote = E_StateRemote.Auto THEN
			// Автоматический режим - динамическая частота от ПИД
			rTargetFreqVibFeeder1 := irManualFrequency; // TODO ВРЕМЕННО Bunker.rMotorVibFeederCommonFrequency
			rTargetFreqVibFeeder2 := irManualFrequency; // TODO ВРЕМЕННО Bunker.rMotorVibFeederCommonFrequency
		ELSE
			// Ручной/Ремонт режим - частота от входного параметра irManualFrequency
			rTargetFreqVibFeeder1 := irManualFrequency;
			rTargetFreqVibFeeder2 := irManualFrequency;
		END_IF;

	E_StageWithPreStartAlarm.ERROR:
		// Состояние ошибки - аварийная остановка и ожидание сброса
		// (используется при серьезных неисправностях, не для штатной остановки)

		// Сброс таймеров
		fbTimerStarting(IN := FALSE);
		fbTimerStopping(IN := FALSE);

		// Аварийная остановка: команда СТОП на VFD (FALSE = СТОП)
		Bunker.MotorVibFeeder[1].VFD.qxStart := FALSE;
		Bunker.MotorVibFeeder[2].VFD.qxStart := FALSE;

		// Сброс целевых частот
		rTargetFreqVibFeeder1 := 0.0;
		rTargetFreqVibFeeder2 := 0.0;

		// Разборка схемы контакторов (аварийная остановка)
//		IF Bunker.eStateRemote = E_StateRemote.Auto THEN
//		 xCircuitBuilt := FALSE;
//		END_IF;
		// Контакторы управляются отдельно через импульсные команды
		// cmdBuildCircuitOn/Off (см. секцию УПРАВЛЕНИЕ КОНТАКТОРАМИ)

		// Сброс ошибки и переход в IDLE при отсутствии ошибок
		// Для выхода из ERROR требуется:
		// 1. Команда сброса (xReset)
		// 2. Снятие сигнала аварийной остановки (NOT xEmergencyStopVibFeeder)
		// 3. Кнопка аварийной остановки отпущена (NC контакт: TRUE = кнопка отпущена)
		// 4. Отсутствие ошибок оборудования (NOT Bunker.xStateFailure)
		IF xReset AND NOT xEmergencyStopVibFeeder AND Bunker.fbBtnEmergencyStop.qxSignal AND NOT Bunker.xStateFailure THEN
			STAGE := E_StageWithPreStartAlarm.IDLE;
		END_IF

END_CASE;

// Выходной параметр - текущая стадия
eStage := STAGE;

// ========================================
// ОБНОВЛЕНИЕ РЕЖИМА УПРАВЛЕНИЯ
// ========================================

// Если установлен местный режим (xLocalMode = TRUE), то переводим в Manual
// Manual может работать как дистанционно (от SCADA), так и местно (от ПМУ)
IF xLocalMode THEN
	Bunker.eStateRemote := E_StateRemote.Manual;
END_IF;

// ========================================
// ОБРАБОТКА ЧАСТОТЫ (после установки целевых значений в CASE)
// ========================================

// Мотор вибропитателя 1
Bunker.MotorVibFeeder[1].VFD.Frequency(
	irMaxFrequency := VFD_FREQUENCY_MAX,
	// Если плавный пуск - используем шаг, иначе - большой шаг для мгновенной установки
	irStep := SEL(VFD_SMOOTH_SET_FREQUENCY, VFD_FREQ_MAX_RANGE, VFD_FREQUENCY_STEP),
	rTargetFrequency := rTargetFreqVibFeeder1,
	xPulse := PULSE_RTRIG.Q,
	xConditionToProceed := TRUE
);
// qrCurrentFrequency передается напрямую в fbAnalogOutput.rEngValue

// Мотор вибропитателя 2
Bunker.MotorVibFeeder[2].VFD.Frequency(
	irMaxFrequency := VFD_FREQUENCY_MAX,
	// Если плавный пуск - используем шаг, иначе - большой шаг для мгновенной установки
	irStep := SEL(VFD_SMOOTH_SET_FREQUENCY, VFD_FREQ_MAX_RANGE, VFD_FREQUENCY_STEP),
	rTargetFrequency := rTargetFreqVibFeeder2,
	xPulse := PULSE_RTRIG.Q,
	xConditionToProceed := TRUE
);
// qrCurrentFrequency передается напрямую в fbAnalogOutput.rEngValue

// ========================================
// ПЕРЕДАЧА СОСТОЯНИЙ ДЛЯ SCADA
// ========================================

// Приоритет проверки: от более критичных к менее критичным
IF STAGE = E_StageWithPreStartAlarm.ERROR THEN
	// Ошибка без активной работы
	eStageToSCADA := E_ScadaStatesDevice.ERROR;

ELSIF STAGE = E_StageWithPreStartAlarm.WORK AND Bunker.xStateFailure THEN
	// TODO: Секция работает с аварией (требует уточнения логики)
	// Обычно при ошибке должна быть остановка, но оставляем для будущей реализации
	eStageToSCADA := E_ScadaStatesDevice.WORK_WITH_ERROR;

ELSIF STAGE = E_StageWithPreStartAlarm.WORK AND Bunker.xStateWarning THEN
	// Секция работает с предупреждением
	eStageToSCADA := E_ScadaStatesDevice.WORK_WITH_WARNING;

ELSIF STAGE = E_StageWithPreStartAlarm.WORK THEN
	// Секция работает в норме (нет ошибок и предупреждений)
	eStageToSCADA := E_ScadaStatesDevice.WORK;

ELSIF STAGE = E_StageWithPreStartAlarm.STARTING THEN
	// Секция в процессе запуска (разгон вибропитателей)
	eStageToSCADA := E_ScadaStatesDevice.STARTING;

ELSIF STAGE = E_StageWithPreStartAlarm.IDLE AND Bunker.xStateWarning THEN
	// Предупреждение без активной работы
	eStageToSCADA := E_ScadaStatesDevice.WARNING;

ELSIF STAGE = E_StageWithPreStartAlarm.IDLE AND Bunker.xStateFailure THEN
	// Секция неготова к запуску (есть ошибки)
	eStageToSCADA := E_ScadaStatesDevice.NOT_READY;

ELSE
	// Секция готова к запуску (IDLE, нет ошибок и предупреждений)
	eStageToSCADA := E_ScadaStatesDevice.READY;

END_IF;

// Передача состояний режима управления вибропитателей
Bunker.xStateRemoteAuto := Bunker.eStateRemote = E_StateRemote.Auto;
Bunker.xStateRemoteManual := Bunker.eStateRemote = E_StateRemote.Manual;
Bunker.xStateRemoteRepair := Bunker.eStateRemote = E_StateRemote.Repair;

// Передача состояний режима управления вибраторов
Bunker.xVibratorStateRemoteAuto := Bunker.eVibratorStateRemote = E_StateRemote.Auto;
Bunker.xVibratorStateRemoteManual := Bunker.eVibratorStateRemote = E_StateRemote.Manual;
Bunker.xVibratorStateRemoteRepair := Bunker.eVibratorStateRemote = E_StateRemote.Repair;

// Передача состояний режима управления светофора
Bunker.xLighterStateRemoteAuto := Bunker.eStateRemoteLighter = E_StateRemote.Auto;
Bunker.xLighterStateRemoteManual := Bunker.eStateRemoteLighter = E_StateRemote.Manual;
Bunker.xLighterStateRemoteRepair := Bunker.eStateRemoteLighter = E_StateRemote.Repair;

// ========================================
// УПРАВЛЕНИЕ КОНТАКТОРАМИ
// ========================================

// РУЧНОЙ РЕЖИМ (Manual):
// - Схема управляется ТОЛЬКО импульсными командами cmdBuildCircuitOn/Off
// - Автоматическая сборка/разборка схемы ОТКЛЮЧЕНА
//
// АВТОМАТИЧЕСКИЙ РЕЖИМ (Auto/Remote):
// - Схема собирается АВТОМАТИЧЕСКИ при отсутствии ошибок секции:
//   * Нет ошибок по оборудованию бункера (FC_Bunker_GetErrorBunker = FALSE)
//   * Секция НЕ в стадии ERROR
// - Схема разбирается АВТОМАТИЧЕСКИ при появлении ошибок или переходе в ERROR

IF Bunker.eStateRemote = E_StateRemote.Manual THEN
	// РУЧНОЙ РЕЖИМ - Обработка импульсных команд сборки/разборки схемы вибропитателей
	// cmdBuildCircuitOn - собрать схему (включить контакторы)
	// cmdBuildCircuitOff - разобрать схему (выключить контакторы)
	IF Bunker.cmdBuildCircuitOn THEN
		xCircuitBuilt := TRUE;
		Bunker.cmdBuildCircuitOn := FALSE; // Сброс импульсной команды
	ELSIF Bunker.cmdBuildCircuitOff THEN
		xCircuitBuilt := FALSE;
		Bunker.cmdBuildCircuitOff := FALSE; // Сброс импульсной команды
	END_IF;
ELSIF Bunker.eStateRemote = E_StateRemote.Auto THEN
	// АВТОМАТИЧЕСКИЙ РЕЖИМ - Автоматическая сборка схемы при отсутствии ошибок
	// Собираем схему если:
	// 1. Нет ошибок по оборудованию бункера (моторы вибропитателей и вибраторов)
	// 2. Секция НЕ в стадии ERROR
	IF NOT FC_Bunker_GetErrorBunker(Bunker := Bunker) AND STAGE <> E_StageWithPreStartAlarm.ERROR AND Bunker.eStateRemote = E_StateRemote.Auto THEN
		xCircuitBuilt := TRUE;
	//ELSE
		//xCircuitBuilt := FALSE;
	END_IF;
END_IF;

// Управление схемой вибраторов
IF Bunker.eVibratorStateRemote = E_StateRemote.Manual THEN
	// РУЧНОЙ РЕЖИМ - Обработка импульсных команд сборки/разборки схемы вибраторов
	// cmdBuildCircuitOnVibrator - собрать схему вибраторов (включить контакторы)
	// cmdBuildCircuitOffVibrator - разобрать схему вибраторов (выключить контакторы)
	IF Bunker.cmdBuildCircuitOnVibrator THEN
		xCircuitBuiltVibrator := TRUE;
		Bunker.cmdBuildCircuitOnVibrator := FALSE; // Сброс импульсной команды
	ELSIF Bunker.cmdBuildCircuitOffVibrator THEN
		xCircuitBuiltVibrator := FALSE;
		Bunker.cmdBuildCircuitOffVibrator := FALSE; // Сброс импульсной команды
	END_IF;
ELSIF Bunker.eVibratorStateRemote = E_StateRemote.Auto THEN
	// АВТОМАТИЧЕСКИЙ РЕЖИМ - Автоматическая сборка схемы вибраторов при отсутствии ошибок
	// Собираем схему если:
	// 1. Нет ошибок по оборудованию бункера (моторы вибропитателей и вибраторов)
	// 2. Секция НЕ в стадии ERROR
	IF NOT FC_Bunker_GetErrorBunker(Bunker := Bunker) AND STAGE <> E_StageWithPreStartAlarm.ERROR THEN
		xCircuitBuiltVibrator := TRUE;
	//ELSE
		//xCircuitBuiltVibrator := FALSE;
	END_IF;
END_IF;

// Моторы вибропитателей - управление контакторами через состояние схемы
Bunker.MotorVibFeeder[1].qxKM_Power := xCircuitBuilt;
Bunker.MotorVibFeeder[2].qxKM_Power := xCircuitBuilt;

// Моторы вибраторов - управление контакторами через состояние схемы
Bunker.MotorVibrator[1].qxKM_Power := xCircuitBuiltVibrator;
Bunker.MotorVibrator[2].qxKM_Power := xCircuitBuiltVibrator;
Bunker.MotorVibrator[3].qxKM_Power := xCircuitBuiltVibrator;
Bunker.MotorVibrator[4].qxKM_Power := xCircuitBuiltVibrator;

// ========================================
// УПРАВЛЕНИЕ РЕЖИМАМИ ВИБРАТОРОВ
// ========================================

// Обработка команд переключения режима управления вибраторов
IF Bunker.cmdVibratorSetModeAuto THEN
	Bunker.eVibratorStateRemote := E_StateRemote.Auto;
	xVibratorManualRunActive := FALSE; // Сброс флага при смене режима
	xVibratorAutoActive := FALSE;
	tonVibratorActive(IN := FALSE);
	tonVibratorPause(IN := FALSE);
ELSIF Bunker.cmdVibratorSetModeManual THEN
	Bunker.eVibratorStateRemote := E_StateRemote.Manual;
	xVibratorManualRunActive := FALSE; // Сброс флага при смене режима
	xVibratorAutoActive := FALSE;
	tonVibratorActive(IN := FALSE);
	tonVibratorPause(IN := FALSE);
ELSIF Bunker.cmdVibratorSetModeRepair THEN
	Bunker.eVibratorStateRemote := E_StateRemote.Repair;
	xVibratorManualRunActive := FALSE; // Сброс флага при смене режима
	xVibratorAutoActive := FALSE;
	tonVibratorActive(IN := FALSE);
	tonVibratorPause(IN := FALSE);
END_IF;

// ========================================
// УПРАВЛЕНИЕ ВИБРАТОРАМИ
// ========================================

// ПРИОРИТЕТНАЯ ПРОВЕРКА АВАРИЙНОЙ ОСТАНОВКИ ВИБРАТОРОВ
// Аварийная остановка вибраторов имеет наивысший приоритет
// При получении сигнала аварийной остановки - немедленная остановка всех вибраторов
IF xEmergencyStopVibrator THEN
	// Остановка всех VFD вибраторов
	Bunker.MotorVibrator[1].VFD.qxStart := FALSE;
	Bunker.MotorVibrator[2].VFD.qxStart := FALSE;
	Bunker.MotorVibrator[3].VFD.qxStart := FALSE;
	Bunker.MotorVibrator[4].VFD.qxStart := FALSE;

	// Разборка схемы контакторов вибраторов
	xCircuitBuiltVibrator := FALSE;

	// Сброс таймеров и флагов
	tonVibratorActive(IN := FALSE);
	tonVibratorPause(IN := FALSE);
	xVibratorManualRunActive := FALSE;
	xVibratorAutoActive := FALSE;
END_IF;

// Нормальная работа вибраторов (если нет аварийной остановки)
IF NOT xEmergencyStopVibrator THEN
	// === РЕЖИМ АВТОМАТИЧЕСКИЙ - циклическая работа по таймеру ===
	IF Bunker.eVibratorStateRemote = E_StateRemote.Auto THEN
		// Автоматический режим работает только в стадии WORK вибропитателей
		IF STAGE = E_StageWithPreStartAlarm.WORK THEN
			// Установка частоты для вибраторов в автоматическом режиме
			FOR i := 1 TO AMOUNT_BUNKER_MOTOR_VIBRATOR BY 1 DO
				Bunker.MotorVibrator[i].VFD.qrOutFrequency := irManualFrequencyVibrator;
			END_FOR;

			// Таймеры автоматического цикла
			tonVibratorActive(PT := VIBRATOR_SETTINGS.TIME_ACTIVE);
			tonVibratorPause(PT := VIBRATOR_SETTINGS.TIME_PAUSE_VIBRATOR);

			// Логика автоматического цикла (ACTIVE → PAUSE → ACTIVE → ...)
			IF NOT xVibratorAutoActive THEN
				// Состояние PAUSE - ждем окончания паузы
				IF tonVibratorPause.Q THEN
					// Пауза завершена - переход в ACTIVE
					tonVibratorPause(IN := FALSE);
					tonVibratorActive(IN := TRUE);
					xVibratorAutoActive := TRUE;

					// Запуск всех вибраторов
					Bunker.MotorVibrator[1].VFD.qxStart := TRUE;
					Bunker.MotorVibrator[2].VFD.qxStart := TRUE;
					Bunker.MotorVibrator[3].VFD.qxStart := TRUE;
					Bunker.MotorVibrator[4].VFD.qxStart := TRUE;
				ELSIF NOT tonVibratorPause.IN THEN
					// Первый запуск - сразу в ACTIVE
					tonVibratorActive(IN := TRUE);
					xVibratorAutoActive := TRUE;

					// Запуск всех вибраторов
					Bunker.MotorVibrator[1].VFD.qxStart := TRUE;
					Bunker.MotorVibrator[2].VFD.qxStart := TRUE;
					Bunker.MotorVibrator[3].VFD.qxStart := TRUE;
					Bunker.MotorVibrator[4].VFD.qxStart := TRUE;
				END_IF;
			ELSE
				// Состояние ACTIVE - ждем окончания активной работы
				IF tonVibratorActive.Q THEN
					// Активная работа завершена - переход в PAUSE
					tonVibratorActive(IN := FALSE);
					tonVibratorPause(IN := TRUE);
					xVibratorAutoActive := FALSE;

					// Остановка всех вибраторов
					Bunker.MotorVibrator[1].VFD.qxStart := FALSE;
					Bunker.MotorVibrator[2].VFD.qxStart := FALSE;
					Bunker.MotorVibrator[3].VFD.qxStart := FALSE;
					Bunker.MotorVibrator[4].VFD.qxStart := FALSE;
				END_IF;
			END_IF;
		ELSE
			// Вне стадии WORK - остановка автоматического цикла
			tonVibratorActive(IN := FALSE);
			tonVibratorPause(IN := FALSE);
			xVibratorAutoActive := FALSE;

			// Остановка всех вибраторов
			Bunker.MotorVibrator[1].VFD.qxStart := FALSE;
			Bunker.MotorVibrator[2].VFD.qxStart := FALSE;
			Bunker.MotorVibrator[3].VFD.qxStart := FALSE;
			Bunker.MotorVibrator[4].VFD.qxStart := FALSE;
		END_IF;

	// === РЕЖИМ РУЧНОЙ - индивидуальное управление через выбор + старт/стоп ===
	ELSIF Bunker.eVibratorStateRemote = E_StateRemote.Manual THEN
		// Команда СТАРТ активирует флаг запуска
		IF Bunker.cmdStartVibrator THEN
			xVibratorManualRunActive := TRUE;
		END_IF

		// Команда СТОП останавливает ВСЕ вибраторы и сбрасывает флаг
		IF Bunker.cmdStopVibrator THEN
			xVibratorManualRunActive := FALSE;
			Bunker.MotorVibrator[1].VFD.qxStart := FALSE;
			Bunker.MotorVibrator[2].VFD.qxStart := FALSE;
			Bunker.MotorVibrator[3].VFD.qxStart := FALSE;
			Bunker.MotorVibrator[4].VFD.qxStart := FALSE;
		END_IF

		// Если флаг запуска активен - управляем вибраторами через галочки выбора
		IF xVibratorManualRunActive THEN
			// Каждый вибратор работает только если он выбран (галочка установлена)
			Bunker.MotorVibrator[1].VFD.qxStart := Bunker.cmdAddVib1;
			Bunker.MotorVibrator[2].VFD.qxStart := Bunker.cmdAddVib2;
			Bunker.MotorVibrator[3].VFD.qxStart := Bunker.cmdAddVib3;
			Bunker.MotorVibrator[4].VFD.qxStart := Bunker.cmdAddVib4;
		END_IF

		// Установка частоты для вибраторов в ручном режиме
		FOR i := 1 TO AMOUNT_BUNKER_MOTOR_VIBRATOR BY 1 DO
			Bunker.MotorVibrator[i].VFD.qrOutFrequency := irManualFrequencyVibrator;
		END_FOR;

	// === РЕЖИМ РЕМОНТ - все вибраторы остановлены ===
	ELSIF Bunker.eVibratorStateRemote = E_StateRemote.Repair THEN
		xVibratorManualRunActive := FALSE;
		xVibratorAutoActive := FALSE;
		Bunker.MotorVibrator[1].VFD.qxStart := FALSE;
		Bunker.MotorVibrator[2].VFD.qxStart := FALSE;
		Bunker.MotorVibrator[3].VFD.qxStart := FALSE;
		Bunker.MotorVibrator[4].VFD.qxStart := FALSE;
	END_IF;
END_IF; // Конец IF NOT xEmergencyStopVibrator

// ========================================
// РУЧНОЕ УПРАВЛЕНИЕ СВЕТОФОРОМ
// ========================================

IF Bunker.eStateRemoteLighter = E_StateRemote.Manual THEN
	// Команда переключения на КРАСНЫЙ
	IF Bunker.cmdLighetSetColorRed THEN FC_Bunker_SetLightColor(Bunker:= Bunker, eColor:= E_LightColor.RED);
	// Команда переключения на ЖЕЛТЫЙ
	ELSIF Bunker.cmdLighetSetColorYellow THEN FC_Bunker_SetLightColor(Bunker:= Bunker, eColor:= E_LightColor.YELLOW);
	// Команда переключения на ЗЕЛЕНЫЙ
	ELSIF Bunker.cmdLighetSetColorGreen THEN FC_Bunker_SetLightColor(Bunker:= Bunker, eColor:= E_LightColor.GREEN);
	// Команда переключения на ВЫКЛЮЧИТЬ
	ELSIF Bunker.cmdLighetSetColorOff THEN FC_Bunker_SetLightColor(Bunker:= Bunker, eColor:= E_LightColor.OFF); END_IF;
END_IF;

// Режим управления АВТО
IF Bunker.cmdLighterSetModeAuto THEN Bunker.eStateRemoteLighter := E_StateRemote.Auto; END_IF;
// Режим управления РУЧНОЙ
IF Bunker.cmdLighterSetModeManual THEN Bunker.eStateRemoteLighter := E_StateRemote.Manual; END_IF;
// Режим управления РЕМОНТ
IF Bunker.cmdLighterSetModeRepair THEN Bunker.eStateRemoteLighter := E_StateRemote.Repair; END_IF;

// ========================================
// РАСЧЁТ ОШИБОК ОБОРУДОВАНИЯ
// ========================================
// Ошибки рассчитываются через отдельные функции FC_Get_ErrorBunker и т.д.

END_FUNCTION_BLOCK

(* ---- FB_ConveyorControl.st ---- *)
FUNCTION_BLOCK FB_ConveyorControl
VAR_INPUT
	Conveyor : REFERENCE TO ST_ConveyorPrefabricated;
	xLocalMode : BOOL; // TRUE = местный режим (ПМУ), FALSE = дистанционный режим (SCADA)
	xStart : BOOL; // Команда запуска конвейера (дистанционный режим)
	xStop : BOOL; // Команда остановки (дистанционный режим)
	xEmergencyStop : BOOL; // Аварийная остановка
	xReset : BOOL; // Сброс в начальное состояние
	xDisableAutoEmergencyStop : BOOL; // Отключение автоматических аварийных остановок по датчикам безопасности
END_VAR
VAR_OUTPUT
	eStage : E_StageWithPreStartAlarm; // Текущая стадия
	eStageToSCADA : E_ScadaStatesDevice; // Передача состояния скаде
END_VAR
VAR
	// Состояния
	STAGE : E_StageWithPreStartAlarm := E_StageWithPreStartAlarm.IDLE;

	// Объединенные команды (ПМУ или SCADA в зависимости от режима)
	xStartCommand : BOOL; // Фактическая команда запуска (из ПМУ или SCADA)
	xStopCommand : BOOL; // Фактическая команда остановки (из ПМУ или SCADA)

	// Подстадии запуска
	nStartingSubstage : INT := 0;
	// 0 - RELEASE_BRAKE, 1 - WAIT_BRAKE_FEEDBACK, 2 - START_VFD, 3 - RAMPING

	// Подстадии остановки
	nStoppingSubstage : INT := 0;
	// 0 - Нормальная работа
	// 1 - SET_FREQUENCY_ZERO: Установка частоты 0 на аналоговый выход
	// 2 - WAIT_FREQUENCY_ZERO: Ожидание подтверждения частоты 0 с аналогового входа
	// 3 - STOP_VFD: Остановка VFD (снятие команды пуска)
	// 4 - WAIT_VFD_STOP: Ожидание остановки VFD (обратная связь)
	// 5 - ACTIVATE_BRAKE: Активация тормозов
	// 6 - WAIT_BRAKE_FEEDBACK: Ожидание обратной связи тормозов

	// Целевые частоты для моторов
	rTargetFreqConv1 : REAL := 0.0;
	rTargetFreqConv2 : REAL := 0.0;

	// Переменные синхронизации моторов конвейера
	xVFDsReady : BOOL; // Оба ЧРП конвейера готовы и запущены
	xFrequenciesSynchronized : BOOL; // Частоты синхронизированы в пределах допуска
	xConditionToProceed : BOOL; // Общее условие для продолжения разгона

	// Состояние схемы контакторов
	xCircuitBuilt : BOOL := FALSE;

	// Таймеры контроля выполнения команд
	fbTimerStarting : TON; // Тайм-аут запуска (STARTING → WORK)
	fbTimerStopping : TON; // Тайм-аут остановки (WORK → IDLE)

	tonTimerEnableBreakerConveyor : TON; // Задержка включения тормоза на конвейере

	simInit : BOOL;
	i : INT;
END_VAR

// ========================================
// FB_ConveyorControl - Управление сборным конвейером
// ========================================
//
// РЕЖИМЫ УПРАВЛЕНИЯ:
//
// 1. МЕСТНЫЙ РЕЖИМ (xLocalMode = TRUE):
//    - Команды берутся с кнопок ПМУ (Conveyor.fbBtnStart, fbBtnStop)
//    - ПУСК/СТОП по фронтам кнопок
//    - Автоматически устанавливает eStateRemote = Manual
//
// 2. ДИСТАНЦИОННЫЙ РЕЖИМ (xLocalMode = FALSE):
//    - Команды берутся из входов ФБ (xStart, xStop)
//    - Режим устанавливается через SCADA (Manual/Remote/Auto)
//
// УПРАВЛЕНИЕ КОНВЕЙЕРОМ:
// - ПУСК: включение конвейеров с предпусковой сигнализацией
// - СТОП: плавная остановка с последовательным выключением VFD и тормозов
//
// ========================================

// ========================================
// ИНИЦИАЛИЗАЦИЯ СИГНАЛОВ
// ========================================

// ПМУ - СТАРТ
Conveyor.fbBtnStart(
	ixSignal := , // Подключить физический вход
	xEnableRattlingFilter := TRUE,
	tStabilityTime := T#100MS
);

// ПМУ - СТОП
Conveyor.fbBtnStop(
	ixSignal := , // Подключить физический вход
	xEnableRattlingFilter := TRUE,
	tStabilityTime := T#100MS
);

// ПМУ - Аварийная остановка
Conveyor.fbBtnEmergencyStop(
	ixSignal := , // Подключить физический вход
	xEnableRattlingFilter := TRUE,
	tStabilityTime := T#100MS
);

// Двигатели конвейера
FOR i := 1 TO 2 BY 1 DO
	Conveyor.MotorConveyor[i].fbStateKM(
		ixSignal := , // Состояние контактора
		xEnableRattlingFilter := TRUE
	);

	Conveyor.MotorConveyor[i].fbStatorOverheat(
		ixSignal := , // Перегрев статора
		xEnableRattlingFilter := TRUE
	);

	Conveyor.MotorConveyor[i].fbStateQF(
		ixSignal := , // Автомат. выключатель
		xEnableRattlingFilter := TRUE
	);

	Conveyor.MotorConveyor[i].VFD.fbStateFailure(
		ixSignal := , // ЧРП - ошибка
		xEnableRattlingFilter := TRUE
	);

	Conveyor.MotorConveyor[i].VFD.fbStateRdyToStart(
		ixSignal := , // ЧРП - Готовность
		xEnableRattlingFilter := TRUE
	);

	Conveyor.MotorConveyor[i].VFD.fbStateIsWorking(
		ixSignal := , // ЧРП - Работа
		xEnableRattlingFilter := TRUE
	);

	// Инициализация устройств
	Conveyor.MotorConveyor[i].Device(
		ixFeedback := Conveyor.MotorConveyor[i].fbStateKM.qxSignal,
		xEnableFeedback := TRUE
	);
	// Контакторы управляются в секции "УПРАВЛЕНИЕ КОНТАКТОРАМИ" через cmdBuildCircuitOn/Off

	// ЧРП
	Conveyor.MotorConveyor[i].VFD.Device(
		ixFeedback := Conveyor.MotorConveyor[i].VFD.fbStateIsWorking.qxSignal,
		xEnableFeedback := TRUE
	);
	// VFD.qxStart теперь управляется напрямую в алгоритме (TRUE = ПУСК, FALSE = СТОП)

	// Диагностика тока
	Conveyor.MotorConveyor[i].VFD.fbRangeDiagnostic(
		irValue := Conveyor.MotorConveyor[i].VFD.wMotorCurrent.rTag,
		irSetpointL := MOTOR_CONVEYOR_CURRENT_POINTS.L_Value,
		irSetpointLL := MOTOR_CONVEYOR_CURRENT_POINTS.LL_Value,
		irSetpointH := MOTOR_CONVEYOR_CURRENT_POINTS.H_Value,
		irSetpointHH := MOTOR_CONVEYOR_CURRENT_POINTS.HH_Value,
		ixEnable := TRUE
	);
	// Аналоговый вход ЧРП (чтение текущей частоты)
	Conveyor.MotorConveyor[i].VFD.fbAnalogInput(
		xSimulation := SIMULATION,
		iADC_Code := Conveyor.MotorConveyor[i].VFD.nActualFrequencyADC,
		refEngValue := Conveyor.MotorConveyor[i].VFD.rActualFrequency,
		refSimValue := Conveyor.MotorConveyor[i].VFD.rSimulatedFrequency,
		rAlarm_LL := VFD_CURRENT_ALARM_LL,
		rAlarm_L := VFD_CURRENT_ALARM_L,
		rAlarm_H := VFD_CURRENT_ALARM_H,
		rAlarm_HH := VFD_CURRENT_ALARM_HH,
		iADC_Max := VFD_ADC_MAX,
		iADC_Min := VFD_ADC_MIN,
		rEngValue_Max := VFD_FREQ_MAX_RANGE,
		rEngValue_Min := VFD_FREQ_MIN,
		rCurrent_Max := VFD_CURRENT_MAX,
		rCurrent_Min := VFD_CURRENT_MIN
	);

	// Аналоговый выход ЧРП (задание частоты)
	Conveyor.MotorConveyor[i].VFD.fbAnalogOutput(
		xEnable := Conveyor.MotorConveyor[i].VFD.fbStateIsWorking.qxSignal,
		rEngValue := Conveyor.MotorConveyor[i].VFD.Frequency.qrCurrentFrequency,
		rEngValue_Max := VFD_FREQ_MAX_RANGE,
		rEngValue_Min := VFD_FREQ_MIN,
		rCurrent_Max := VFD_CURRENT_MAX,
		rCurrent_Min := VFD_CURRENT_MIN,
		iDAC_Max := VFD_ADC_MAX,
		iDAC_Min := VFD_ADC_MIN,
		rAlarm_LL := VFD_CURRENT_ALARM_LL,
		rAlarm_L := VFD_CURRENT_ALARM_L,
		rAlarm_H := VFD_CURRENT_ALARM_H,
		rAlarm_HH := VFD_CURRENT_ALARM_HH,
		xEnableClamp := TRUE
	);
	Conveyor.MotorConveyor[i].VFD.nSetOutSignalToModule := Conveyor.MotorConveyor[i].VFD.fbAnalogOutput.iDAC_Code;
END_FOR;

// Датчики безопасности
FOR i := 1 TO 4 BY 1 DO
	Conveyor.fbZQAlarm[i](
		ixSignal := ,
		xEnableRattlingFilter := TRUE
	);

	Conveyor.fbZQWarning[i](
		ixSignal := ,
		xEnableRattlingFilter := TRUE
	);

	Conveyor.fbHQ_IsOk[i](
		ixSignal := ,
		xEnableRattlingFilter := TRUE
	);
END_FOR;

FOR i := 1 TO 2 BY 1 DO
	Conveyor.fbSQ_IsOk[i](
		ixSignal := ,
		xEnableRattlingFilter := TRUE
	);

	Conveyor.fbQR[i](
		ixSignal := ,
		xEnableRattlingFilter := FALSE // Только edge detection
	);
END_FOR;

Conveyor.fbGS1(
	ixSignal := ,
	xEnableRattlingFilter := TRUE
);

Conveyor.fbYS1(
	ixSignal := ,
	xEnableRattlingFilter := TRUE
);

Conveyor.fbYE1(
	ixSignal := ,
	xEnableRattlingFilter := TRUE
);

// Обратная связь тормоза конвейера
Conveyor.fbBreakerConveyor(
	ixSignal := , // Обратная связь реле тормоза
	xEnableRattlingFilter := TRUE
);

// ========================================
// ПРЕДПУСКОВАЯ СИГНАЛИЗАЦИЯ
// ========================================

Conveyor.fbPreStartAlarm(
	ixStart := STAGE = PRESTART_ALARM,
	ixStop := xStopCommand OR xReset,
	itFirstSignal := CONVEYOR_PRESTART_ALARM_SETTINGS.TIME_FIRST_SIGNAL,
	itPauseAfterFirst := CONVEYOR_PRESTART_ALARM_SETTINGS.TIME_FIRST_SIGNAL_PAUSE,
	itSecondSignal := CONVEYOR_PRESTART_ALARM_SETTINGS.TIME_SECOND_SIGNAL,
	itPauseAfterSecond := CONVEYOR_PRESTART_ALARM_SETTINGS.TIME_SECOND_SIGNAL_PAUSE,
	qxAlarmPower => Conveyor.xHLA
);

Conveyor.xStateEnable := STAGE = E_StageWithPreStartAlarm.WORK;
Conveyor.xStateStarting := STAGE = E_StageWithPreStartAlarm.STARTING OR STAGE = PRESTART_ALARM;

// ========================================
// ОПРЕДЕЛЕНИЕ СОСТОЯНИЙ ДЛЯ SCADA
// ========================================

// Проверка ошибок оборудования
IF FC_Conveyor_GetErrorCommon(Conveyor := Conveyor) OR fbTimerStarting.Q THEN
	Conveyor.xStateFailure := TRUE;
END_IF;

// Проверка предупреждений:
// 1. Датчики схода ленты ZQ - уровень Warning
// 2. Контроль тока моторов - уровень L или H
Conveyor.xStateWarning := NOT Conveyor.fbZQWarning[1].qxSignal
                       OR NOT Conveyor.fbZQWarning[2].qxSignal
                       OR NOT Conveyor.fbZQWarning[3].qxSignal
                       OR NOT Conveyor.fbZQWarning[4].qxSignal
                       OR Conveyor.MotorConveyor[1].VFD.fbRangeDiagnostic.qxWarningActive
                       OR Conveyor.MotorConveyor[2].VFD.fbRangeDiagnostic.qxWarningActive;

// ========================================
// ОБРАБОТКА ОСТАНОВКИ И СБРОСА
// ========================================

// Сброс в начальное состояние
IF xReset THEN
	Conveyor.xStateFailure := FALSE;
END_IF

// ========================================
// ВЫБОР ИСТОЧНИКА КОМАНД (ПМУ ИЛИ SCADA)
// ========================================

// В местном режиме (xLocalMode = TRUE) - команды берутся с ПМУ (кнопки)
// В дистанционном режиме (xLocalMode = FALSE) - команды берутся из SCADA (входы ФБ)
IF xLocalMode THEN
	// Местный режим - команды с ПМУ
	xStartCommand := Conveyor.fbBtnStart.qxRisingEdge; // ПУСК по фронту кнопки
	xStopCommand := Conveyor.fbBtnStop.qxRisingEdge;   // СТОП по фронту кнопки
ELSE
	// Дистанционный режим - команды из SCADA
	xStartCommand := xStart;
	xStopCommand := xStop;
END_IF;

// ========================================
// АВТОМАТ ПУСКА КОНВЕЙЕРА
// ========================================

// ПРИОРИТЕТНАЯ ПРОВЕРКА АВАРИЙНОЙ ОСТАНОВКИ
// Аварийная остановка имеет наивысший приоритет и срабатывает в любой стадии
// 1. Внешний сигнал аварийной остановки (от SCADA или системы)
// 2. Кнопка аварийной остановки на ПМУ (NC контакт: FALSE = кнопка нажата)
IF xEmergencyStop OR NOT Conveyor.fbBtnEmergencyStop.qxSignal THEN
	STAGE := E_StageWithPreStartAlarm.ERROR;
END_IF;

// КРИТИЧЕСКИЕ ОШИБКИ ДАТЧИКОВ БЕЗОПАСНОСТИ
// При срабатывании датчиков безопасности немедленная аварийная остановка,
// если секция НЕ в IDLE (т.е. находится в процессе работы или запуска)
// Блокируется через вход xDisableAutoEmergencyStop
IF FC_Conveyor_GetErrorSensors(Conveyor := Conveyor)
   AND STAGE <> E_StageWithPreStartAlarm.IDLE
   AND NOT xDisableAutoEmergencyStop
THEN
	STAGE := E_StageWithPreStartAlarm.ERROR;
END_IF;

// ПРОВЕРКА ТАЙМ-АУТОВ ВЫПОЛНЕНИЯ КОМАНД
// Тайм-аут запуска: не удалось запустить секцию за установленное время
IF fbTimerStarting.Q THEN
	STAGE := E_StageWithPreStartAlarm.ERROR;
END_IF;

// Тайм-аут остановки: не удалось остановить секцию за установленное время
IF fbTimerStopping.Q THEN
	STAGE := E_StageWithPreStartAlarm.ERROR;
END_IF;

CASE STAGE OF
	E_StageWithPreStartAlarm.IDLE:
		// Установка тормозов в активное состояние (FALSE = тормоз активен)
		Conveyor.qxBreakerConveyor := FALSE;

		// Сброс целевой частоты
		rTargetFreqConv1 := 0.0;
		rTargetFreqConv2 := 0.0;

		// Сброс подстадий
		nStartingSubstage := 0;
		nStoppingSubstage := 0;

		// Сброс таймеров запуска и остановки
		fbTimerStarting(IN := FALSE);
		fbTimerStopping(IN := FALSE);

		IF xStartCommand THEN
			STAGE := PRESTART_ALARM;
		END_IF;

	E_StageWithPreStartAlarm.PRESTART_ALARM:
		// Проверка команды остановки во время предпусковой сигнализации
		IF xStopCommand THEN
			// Прервать предпусковую сигнализацию и вернуться в IDLE
			STAGE := E_StageWithPreStartAlarm.IDLE;
		ELSIF Conveyor.fbPreStartAlarm.qxComplete THEN
			STAGE := E_StageWithPreStartAlarm.STARTING;
		END_IF;

	E_StageWithPreStartAlarm.STARTING:
		// Проверка команды остановки во время запуска
		IF xStopCommand THEN
			// Прервать запуск и перейти к процедуре остановки
			STAGE := E_StageWithPreStartAlarm.WORK;
			nStartingSubstage := 0;
			nStoppingSubstage := 1; // Начать процедуру остановки
			fbTimerStarting(IN := FALSE); // Сброс таймера
		END_IF;

		// Таймер ожидания полного запуска секции
		fbTimerStarting(
			IN := TRUE,
			PT := TIME_AFTER_START_CONVEYOR
		);
		CASE nStartingSubstage OF
			0: // RELEASE_BRAKE - Отпускание тормозов
				// Отпускаем тормоз конвейера (TRUE = тормоз отпущен)
				Conveyor.qxBreakerConveyor := TRUE;
				nStartingSubstage := 1;

			1: // WAIT_BRAKE_FEEDBACK - Ожидание обратной связи тормоза
				IF Conveyor.fbBreakerConveyor.qxSignal THEN
					nStartingSubstage := 2;
				END_IF;

			2: // START_VFD - Запуск VFD
				// Команда ПУСК на ЧРП (TRUE = ПУСК)
				Conveyor.MotorConveyor[1].VFD.qxStart := TRUE;
				Conveyor.MotorConveyor[2].VFD.qxStart := TRUE;

				// Задание целевой частоты
				rTargetFreqConv1 := MOTOR_FREQUENCY_CONVEYOR;
				rTargetFreqConv2 := MOTOR_FREQUENCY_CONVEYOR;

				// Ждем запуска ЧРП
				IF Conveyor.MotorConveyor[1].VFD.fbStateIsWorking.qxSignal
					AND Conveyor.MotorConveyor[2].VFD.fbStateIsWorking.qxSignal
				THEN
					IF VFD_SMOOTH_SET_FREQUENCY THEN
						nStartingSubstage := 3; // Плавный разгон
					ELSE
						STAGE := E_StageWithPreStartAlarm.WORK; // Прямой пуск
						nStartingSubstage := 0;
						fbTimerStarting(IN := FALSE); // Сброс таймера
					END_IF;
				END_IF;

			3: // RAMPING - Разгон частоты до рабочей
				// Продолжаем удерживать команду ПУСК на ЧРП
				Conveyor.MotorConveyor[1].VFD.qxStart := TRUE;
				Conveyor.MotorConveyor[2].VFD.qxStart := TRUE;

				// Задание целевой частоты
				rTargetFreqConv1 := MOTOR_FREQUENCY_CONVEYOR;
				rTargetFreqConv2 := MOTOR_FREQUENCY_CONVEYOR;

				// Переход в режим WORK при достижении целевой частоты
				IF Conveyor.MotorConveyor[1].VFD.rActualFrequency >= MOTOR_FREQUENCY_CONVEYOR - VFD_FREQUENCY_INACCURANCY
					AND Conveyor.MotorConveyor[2].VFD.rActualFrequency >= MOTOR_FREQUENCY_CONVEYOR - VFD_FREQUENCY_INACCURANCY
				THEN
					STAGE := E_StageWithPreStartAlarm.WORK;
					nStartingSubstage := 0;
					fbTimerStarting(IN := FALSE); // Сброс таймера
				END_IF;
		END_CASE;

	E_StageWithPreStartAlarm.WORK:
		CASE nStoppingSubstage OF
			0: // Нормальная работа
				// Сброс таймера остановки
				fbTimerStopping(IN := FALSE);

				// Обновление целевой частоты конвейера в ручном режиме
				IF Conveyor.eStateRemote = E_StateRemote.Manual THEN
					rTargetFreqConv1 := MOTOR_FREQUENCY_CONVEYOR;
					rTargetFreqConv2 := MOTOR_FREQUENCY_CONVEYOR;
				END_IF;

				// Проверка команды остановки
				IF xStopCommand THEN
					nStoppingSubstage := 1;
				END_IF;

			1: // SET_FREQUENCY_ZERO - Установка частоты 0 на аналоговый выход
				// Запуск таймера остановки (тайм-аут на остановку секции)
				fbTimerStopping(
					IN := TRUE,
					PT := TIME_TIMEOUT_STOP_CONVEYOR
				);

				// Установить целевую частоту 0
				// (FB_FrequencyControl автоматически выберет плавную или прямую остановку через irStep)
				rTargetFreqConv1 := 0.0;
				rTargetFreqConv2 := 0.0;

				// Команды пуска VFD остаются активными (TRUE = ПУСК)
				// VFD продолжают работать, но частота снижается
				Conveyor.MotorConveyor[1].VFD.qxStart := FALSE; // TODO ВРЕМЕННО
				Conveyor.MotorConveyor[2].VFD.qxStart := FALSE;

				// Переход к следующей подстадии
				nStoppingSubstage := 2;

			2: // WAIT_FREQUENCY_ZERO - Ожидание подтверждения частоты 0 с аналогового входа
				// Ждём, пока фактическая частота (с аналогового входа) не снизится до 0 (+/- 2 Гц)
				IF Conveyor.MotorConveyor[1].VFD.rActualFrequency <= 2.0
					AND Conveyor.MotorConveyor[2].VFD.rActualFrequency <= 2.0
				THEN
					// Частота подтверждена на 0, переходим к остановке VFD
					nStoppingSubstage := 3;
				END_IF;

			3: // STOP_VFD - Остановка VFD (снятие команды пуска)
				// Отключить команду пуска на VFD (FALSE = СТОП)
				Conveyor.MotorConveyor[1].VFD.qxStart := FALSE;
				Conveyor.MotorConveyor[2].VFD.qxStart := FALSE;

				// Переход к ожиданию обратной связи VFD
				nStoppingSubstage := 4;

			4: // WAIT_VFD_STOP - Ожидание остановки VFD (обратная связь)
				// Проверить обратную связь VFD о выключении
				IF NOT Conveyor.MotorConveyor[1].VFD.fbStateIsWorking.qxSignal
					AND NOT Conveyor.MotorConveyor[2].VFD.fbStateIsWorking.qxSignal
				THEN
					// VFD выключены, переход к активации тормозов
					nStoppingSubstage := 5;
				END_IF;

			5: // ACTIVATE_BRAKE - Активация тормозов
				tonTimerEnableBreakerConveyor(IN:= TRUE, PT:=T#5S);
				IF tonTimerEnableBreakerConveyor.Q THEN
					// Снять сигнал с тормоза (поставить на тормоз: FALSE = активен)
					Conveyor.qxBreakerConveyor := FALSE;
					// Переход к завершению остановки
					tonTimerEnableBreakerConveyor(IN:=  FALSE);
					nStoppingSubstage := 6;
				END_IF;
			6: // WAIT_BRAKE_FEEDBACK - Переход в IDLE
				// Сброс таймера остановки (успешная остановка)
				fbTimerStopping(IN := FALSE);

				STAGE := E_StageWithPreStartAlarm.IDLE;
				nStoppingSubstage := 0;
		END_CASE;

	E_StageWithPreStartAlarm.ERROR:
		// Состояние ошибки - аварийная остановка и ожидание сброса
		// (используется при серьезных неисправностях, не для штатной остановки)

		// Аварийная остановка: команда СТОП на VFD (FALSE = СТОП)
		Conveyor.MotorConveyor[1].VFD.qxStart := FALSE;
		Conveyor.MotorConveyor[2].VFD.qxStart := FALSE;

		// Сброс целевых частот
		rTargetFreqConv1 := 0.0;
		rTargetFreqConv2 := 0.0;

		// Активировать тормоз
		Conveyor.qxBreakerConveyor := FALSE;

		// Разборка схемы контакторов (аварийная остановка)
		IF Conveyor.eStateRemote = E_StateRemote.Auto THEN
			xCircuitBuilt := FALSE;
		END_IF;

		// Сброс подстадий для следующего запуска
		nStartingSubstage := 0;
		nStoppingSubstage := 0;

		// Сброс таймеров
		fbTimerStarting(IN := FALSE);
		fbTimerStopping(IN := FALSE);

		// Контакторы управляются отдельно через импульсные команды
		// cmdBuildCircuitOn/Off (см. секцию УПРАВЛЕНИЕ КОНТАКТОРАМИ)

		// Сброс ошибки и переход в IDLE при отсутствии ошибок
		// Для выхода из ERROR требуется:
		// 1. Команда сброса (xReset)
		// 2. Снятие сигнала аварийной остановки (NOT xEmergencyStop)
		// 3. Кнопка аварийной остановки отпущена (NC контакт: TRUE = кнопка отпущена)
		// 4. Отсутствие ошибок оборудования (NOT Conveyor.xStateFailure)
		IF xReset AND NOT xEmergencyStop AND Conveyor.fbBtnEmergencyStop.qxSignal AND NOT Conveyor.xStateFailure THEN
			STAGE := E_StageWithPreStartAlarm.IDLE;
		END_IF
END_CASE;

// Вывод текущей стадии
eStage := STAGE;

// ========================================
// ОБНОВЛЕНИЕ РЕЖИМА УПРАВЛЕНИЯ
// ========================================

// Если установлен местный режим (xLocalMode = TRUE), то переводим в Manual
// Manual может работать как дистанционно (от SCADA), так и местно (от ПМУ)
IF xLocalMode THEN
	Conveyor.eStateRemote := E_StateRemote.Manual;
END_IF;

// ========================================
// ПЕРЕДАЧА СОСТОЯНИЙ ДЛЯ SCADA
// ========================================

// Приоритет проверки: от более критичных к менее критичным
IF STAGE = E_StageWithPreStartAlarm.ERROR THEN
	// Ошибка без активной работы
	eStageToSCADA := E_ScadaStatesDevice.ERROR;

ELSIF STAGE = E_StageWithPreStartAlarm.WORK AND Conveyor.xStateFailure THEN
	// TODO: Секция работает с аварией (требует уточнения логики)
	// Обычно при ошибке должна быть остановка, но оставляем для будущей реализации
	eStageToSCADA := E_ScadaStatesDevice.WORK_WITH_ERROR;

ELSIF STAGE = E_StageWithPreStartAlarm.WORK AND Conveyor.xStateWarning THEN
	// Секция работает с предупреждением
	eStageToSCADA := E_ScadaStatesDevice.WORK_WITH_WARNING;

ELSIF STAGE = E_StageWithPreStartAlarm.WORK THEN
	// Секция работает в норме (нет ошибок и предупреждений)
	eStageToSCADA := E_ScadaStatesDevice.WORK;

ELSIF Conveyor.xStateStarting THEN
	// Секция в процессе запуска (предпусковая сигнализация или разгон)
	eStageToSCADA := E_ScadaStatesDevice.STARTING;

ELSIF STAGE = E_StageWithPreStartAlarm.IDLE AND Conveyor.xStateWarning THEN
	// Предупреждение без активной работы
	eStageToSCADA := E_ScadaStatesDevice.WARNING;

ELSIF STAGE = E_StageWithPreStartAlarm.IDLE AND Conveyor.xStateFailure THEN
	// Секция неготова к запуску (есть ошибки)
	eStageToSCADA := E_ScadaStatesDevice.NOT_READY;

ELSE
	// Секция готова к запуску (IDLE, нет ошибок и предупреждений)
	eStageToSCADA := E_ScadaStatesDevice.READY;

END_IF;

// Передача состояний режима управления
Conveyor.xStateRemoteAuto := Conveyor.eStateRemote = E_StateRemote.Auto;
Conveyor.xStateRemoteManual := Conveyor.eStateRemote = E_StateRemote.Manual;
Conveyor.xStateRemoteRepair := Conveyor.eStateRemote = E_StateRemote.Repair;

// ========================================
// ПРОВЕРКА СИНХРОНИЗАЦИИ МОТОРОВ КОНВЕЙЕРА
// ========================================

// Проверка что оба ЧРП конвейера готовы и запущены
xVFDsReady := Conveyor.MotorConveyor[1].VFD.fbStateIsWorking.qxSignal
           AND Conveyor.MotorConveyor[2].VFD.fbStateIsWorking.qxSignal;

// Проверка синхронизации текущих частот (разница не превышает допуск)
xFrequenciesSynchronized := ABS(Conveyor.MotorConveyor[1].VFD.Frequency.qrCurrentFrequency
                              - Conveyor.MotorConveyor[2].VFD.Frequency.qrCurrentFrequency)
                              <= VFD_FREQUENCY_SYNC_TOLERANCE;

// Общее условие для продолжения плавного разгона
// Разгон продолжается только если оба ЧРП запущены И частоты синхронизированы
xConditionToProceed := xVFDsReady AND xFrequenciesSynchronized;

// ========================================
// ОБРАБОТКА ЧАСТОТЫ (после установки целевых значений в CASE)
// ========================================

// Моторы конвейера
Conveyor.MotorConveyor[1].VFD.Frequency(
	irMaxFrequency := VFD_FREQUENCY_MAX,
	// Если плавный пуск - малый шаг, иначе - большой шаг (мгновенно)
	irStep := SEL(VFD_SMOOTH_SET_FREQUENCY, VFD_FREQ_MAX_RANGE, VFD_FREQUENCY_STEP),
	rTargetFrequency := rTargetFreqConv1,
	xPulse := PULSE_RTRIG.Q,
	xConditionToProceed := xConditionToProceed // Синхронизация с мотором 2
);

Conveyor.MotorConveyor[2].VFD.Frequency(
	irMaxFrequency := VFD_FREQUENCY_MAX,
	// Если плавный пуск - малый шаг, иначе - большой шаг (мгновенно)
	irStep := SEL(VFD_SMOOTH_SET_FREQUENCY, VFD_FREQ_MAX_RANGE, VFD_FREQUENCY_STEP),
	rTargetFrequency := rTargetFreqConv2,
	xPulse := PULSE_RTRIG.Q,
	xConditionToProceed := xConditionToProceed // Синхронизация с мотором 1
);

// ========================================
// УПРАВЛЕНИЕ КОНТАКТОРАМИ
// ========================================

// РУЧНОЙ РЕЖИМ (Manual):
// - Схема управляется ТОЛЬКО импульсными командами cmdBuildCircuitOn/Off
// - Автоматическая сборка/разборка схемы ОТКЛЮЧЕНА
//
// АВТОМАТИЧЕСКИЙ РЕЖИМ (Auto/Remote):
// - Схема собирается АВТОМАТИЧЕСКИ при отсутствии ошибок секции:
//   * Нет ошибок по датчикам безопасности (FC_Conveyor_GetErrorSensors = FALSE)
//   * Секция НЕ в стадии ERROR
// - Схема разбирается АВТОМАТИЧЕСКИ при появлении ошибок или переходе в ERROR

IF Conveyor.eStateRemote = E_StateRemote.Manual THEN
	// РУЧНОЙ РЕЖИМ - Обработка импульсных команд сборки/разборки схемы
	// cmdBuildCircuitOn - собрать схему (включить контакторы)
	// cmdBuildCircuitOff - разобрать схему (выключить контакторы)
	IF Conveyor.cmdBuildCircuitOn THEN
		xCircuitBuilt := TRUE;
		Conveyor.cmdBuildCircuitOn := FALSE; // Сброс импульсной команды
	ELSIF Conveyor.cmdBuildCircuitOff THEN
		xCircuitBuilt := FALSE;
		Conveyor.cmdBuildCircuitOff := FALSE; // Сброс импульсной команды
	END_IF;
ELSIF Conveyor.eStateRemote = E_StateRemote.Auto THEN
	// АВТОМАТИЧЕСКИЙ РЕЖИМ - Автоматическая сборка схемы при отсутствии ошибок
	// Собираем схему если:
	// 1. Нет ошибок по датчикам безопасности
	// 2. Секция НЕ в стадии ERROR
	IF NOT FC_Conveyor_GetErrorSensors(Conveyor := Conveyor) AND STAGE <> E_StageWithPreStartAlarm.ERROR THEN
		xCircuitBuilt := TRUE;
	ELSE
		xCircuitBuilt := FALSE;
	END_IF;
END_IF;

// Моторы конвейера - управление контакторами через состояние схемы
Conveyor.MotorConveyor[1].qxKM_Power := xCircuitBuilt;
Conveyor.MotorConveyor[2].qxKM_Power := xCircuitBuilt;

END_FUNCTION_BLOCK

(* ---- FB_ConveyorWeight.st ---- *)
FUNCTION_BLOCK FB_ConveyorWeight
VAR_INPUT
	wModbusReg : ARRAY [0..22] OF WORD;
END_VAR
VAR_OUTPUT
	qrWeight : REAL; 			//	0x0 Производительность
	qrSpeed : REAL; 			//	0x2 Скорость
	qrWorkLoad : REAL; 			//	0x4 Погонная нагрузка
	qrVoltageTenso_1 : REAL; 	//	0x6 Текущее напряжение тензодатчика 1
	qrVoltageTenso_2 : REAL; 	//	0x8 Текущее напряжение тензодатчика 2
	qrVoltageTenso_3 : REAL; 	//	0xA Текущее напряжение тензодатчика 3
	qrVoltageTenso_4 : REAL; 	//	0xC Текущее напряжение тензодатчика 4
 	qrCounterShift : REAL;		//	0xE Счётчик: смена
	qrCounterDay : REAL;		//	0xE Счётчик: смена
	qrCounterMonth : REAL;		//	0xE Счётчик: смена
	qrCounterCommon : REAL;		//	0xE Счётчик: смена

END_VAR
VAR
END_VAR

END_FUNCTION_BLOCK

(* ---- FB_EmergencyStopProcess.st ---- *)
FUNCTION_BLOCK FB_EmergencyStopProcess
VAR_INPUT
	ixEnable : BOOL;
	ixReset : BOOL;

	Bunker : REFERENCE TO ARRAY [1..3] OF ST_Bunker;
	Dumper : REFERENCE TO ST_Dumper;
	Conveyor : REFERENCE TO ST_ConveyorPrefabricated;
END_VAR
VAR_OUTPUT
	qxStateStopProcess : BOOL;
	qxStateEmergencyStop : BOOL;
	qnCurrentStage : INT;
END_VAR
VAR
	i, j : INT;
	xBunkersStopped : BOOL;
	xConveyorStopped : BOOL;
	xDumperStopped : BOOL;
END_VAR

// Сброс процесса аварийной остановки
IF ixReset THEN
	qxStateStopProcess := FALSE;
	qxStateEmergencyStop := FALSE;
	qnCurrentStage := 0;
	RETURN;
END_IF

// Запуск процесса аварийной остановки
IF ixEnable AND NOT qxStateEmergencyStop AND qnCurrentStage = 0 THEN
	qxStateStopProcess := TRUE;
	qnCurrentStage := 1; // Начинаем с остановки бункеров
END_IF

CASE qnCurrentStage OF

	// === ЭТАП 1: Остановка бункеров ===
	1:
		// Отправляем команды остановки
		FOR i := 1 TO 3 DO
			// Остановка моторов вибраторов (4 шт на бункер)
			FOR j := 1 TO 4 DO
				Bunker[i].MotorVibrator[j].qxKM_Power := FALSE;
				Bunker[i].MotorVibrator[j].VFD.qxStart := FALSE;
				Bunker[i].MotorVibrator[j].VFD.Frequency.rTargetFrequency := 0.0;
				Bunker[i].MotorVibrator[j].VFD.qrOutFrequency := 0.0;
			END_FOR

			// Остановка моторов вибропитателей (2 шт на бункер)
			FOR j := 1 TO 2 DO
				Bunker[i].MotorVibFeeder[j].qxKM_Power := FALSE;
				Bunker[i].MotorVibFeeder[j].VFD.qxStart := FALSE;
				Bunker[i].MotorVibFeeder[j].VFD.Frequency.rTargetFrequency := 0.0;
				Bunker[i].MotorVibFeeder[j].VFD.qrOutFrequency := 0.0;
			END_FOR

			// Установка красного сигнала светофора
			FC_Bunker_SetLightColor(Bunker := Bunker[i], eColor := E_LightColor.RED);
		END_FOR

		// Проверка обратной связи - все моторы бункеров остановлены
		// Используем проверку через прямое вычисление результата
		xBunkersStopped :=
			// Бункер 1
			NOT Bunker[1].MotorVibrator[1].fbStateKM.qxSignal AND NOT Bunker[1].MotorVibrator[1].VFD.xStateIsWorking
			AND NOT Bunker[1].MotorVibrator[2].fbStateKM.qxSignal AND NOT Bunker[1].MotorVibrator[2].VFD.xStateIsWorking
			AND NOT Bunker[1].MotorVibrator[3].fbStateKM.qxSignal AND NOT Bunker[1].MotorVibrator[3].VFD.xStateIsWorking
			AND NOT Bunker[1].MotorVibrator[4].fbStateKM.qxSignal AND NOT Bunker[1].MotorVibrator[4].VFD.xStateIsWorking
			AND NOT Bunker[1].MotorVibFeeder[1].fbStateKM.qxSignal AND NOT Bunker[1].MotorVibFeeder[1].VFD.xStateIsWorking
			AND NOT Bunker[1].MotorVibFeeder[2].fbStateKM.qxSignal AND NOT Bunker[1].MotorVibFeeder[2].VFD.xStateIsWorking
			// Бункер 2
			AND NOT Bunker[2].MotorVibrator[1].fbStateKM.qxSignal AND NOT Bunker[2].MotorVibrator[1].VFD.xStateIsWorking
			AND NOT Bunker[2].MotorVibrator[2].fbStateKM.qxSignal AND NOT Bunker[2].MotorVibrator[2].VFD.xStateIsWorking
			AND NOT Bunker[2].MotorVibrator[3].fbStateKM.qxSignal AND NOT Bunker[2].MotorVibrator[3].VFD.xStateIsWorking
			AND NOT Bunker[2].MotorVibrator[4].fbStateKM.qxSignal AND NOT Bunker[2].MotorVibrator[4].VFD.xStateIsWorking
			AND NOT Bunker[2].MotorVibFeeder[1].fbStateKM.qxSignal AND NOT Bunker[2].MotorVibFeeder[1].VFD.xStateIsWorking
			AND NOT Bunker[2].MotorVibFeeder[2].fbStateKM.qxSignal AND NOT Bunker[2].MotorVibFeeder[2].VFD.xStateIsWorking
			// Бункер 3
			AND NOT Bunker[3].MotorVibrator[1].fbStateKM.qxSignal AND NOT Bunker[3].MotorVibrator[1].VFD.xStateIsWorking
			AND NOT Bunker[3].MotorVibrator[2].fbStateKM.qxSignal AND NOT Bunker[3].MotorVibrator[2].VFD.xStateIsWorking
			AND NOT Bunker[3].MotorVibrator[3].fbStateKM.qxSignal AND NOT Bunker[3].MotorVibrator[3].VFD.xStateIsWorking
			AND NOT Bunker[3].MotorVibrator[4].fbStateKM.qxSignal AND NOT Bunker[3].MotorVibrator[4].VFD.xStateIsWorking
			AND NOT Bunker[3].MotorVibFeeder[1].fbStateKM.qxSignal AND NOT Bunker[3].MotorVibFeeder[1].VFD.xStateIsWorking
			AND NOT Bunker[3].MotorVibFeeder[2].fbStateKM.qxSignal AND NOT Bunker[3].MotorVibFeeder[2].VFD.xStateIsWorking;

		// Переход к следующему этапу
		IF xBunkersStopped THEN
			qnCurrentStage := 2;
		END_IF

	// === ЭТАП 2: Остановка конвейера ===
	2:
		// Отправляем команды остановки
		FOR j := 1 TO 2 DO
			Conveyor.MotorConveyor[j].qxKM_Power := FALSE;
			Conveyor.MotorConveyor[j].VFD.qxStart := FALSE;
			Conveyor.MotorConveyor[j].VFD.Frequency.rTargetFrequency := 0.0;
			Conveyor.MotorConveyor[j].VFD.qrOutFrequency := 0.0;
		END_FOR

		// Проверка обратной связи - моторы конвейера остановлены и процесс запуска не активен
		xConveyorStopped :=
			NOT Conveyor.MotorConveyor[1].fbStateKM.qxSignal AND NOT Conveyor.MotorConveyor[1].VFD.xStateIsWorking
			AND NOT Conveyor.MotorConveyor[2].fbStateKM.qxSignal AND NOT Conveyor.MotorConveyor[2].VFD.xStateIsWorking
			AND NOT Conveyor.xStateStarting; // Добавлена проверка что процесс запуска остановлен

		// Переход к следующему этапу
		IF xConveyorStopped THEN
			qnCurrentStage := 3;
		END_IF

	// === ЭТАП 3: Остановка отвалообразователя ===
	3:
		// Остановка моторов конвейера (унаследовано от ST_ConveyorBasic)
		FOR j := 1 TO 2 DO
			Dumper.MotorConveyor[j].qxKM_Power := FALSE;
			Dumper.MotorConveyor[j].VFD.qxStart := FALSE;
			Dumper.MotorConveyor[j].VFD.Frequency.rTargetFrequency := 0.0;
			Dumper.MotorConveyor[j].VFD.qrOutFrequency := 0.0;
		END_FOR

		// Остановка моторов поворота
		FOR j := 1 TO 2 DO
			Dumper.MotorRotation[j].qxKM_Power := FALSE;
			Dumper.MotorRotation[j].VFD.qxStart := FALSE;
			Dumper.MotorRotation[j].VFD.Frequency.rTargetFrequency := 0.0;
			Dumper.MotorRotation[j].VFD.qrOutFrequency := 0.0;
			Dumper.MotorRotation[j].qxVFDReverseStart := FALSE;
		END_FOR

		// Проверка обратной связи - все моторы отвалообразователя остановлены и процесс запуска не активен
		xDumperStopped :=
			// Моторы конвейера
			NOT Dumper.MotorConveyor[1].fbStateKM.qxSignal AND NOT Dumper.MotorConveyor[1].VFD.xStateIsWorking
			AND NOT Dumper.MotorConveyor[2].fbStateKM.qxSignal AND NOT Dumper.MotorConveyor[2].VFD.xStateIsWorking
			// Моторы поворота
			AND NOT Dumper.MotorRotation[1].fbStateKM.qxSignal AND NOT Dumper.MotorRotation[1].VFD.xStateIsWorking
			AND NOT Dumper.MotorRotation[2].fbStateKM.qxSignal AND NOT Dumper.MotorRotation[2].VFD.xStateIsWorking
			// Проверка что процесс запуска остановлен
			AND NOT Dumper.xStateStarting;

		// Переход к завершению
		IF xDumperStopped THEN
			qnCurrentStage := 4;
		END_IF

	// === ЭТАП 4: Завершение ===
	4:
		qxStateStopProcess := FALSE;
		qxStateEmergencyStop := TRUE;
		// Остаёмся в этом состоянии до ресета

END_CASE

END_FUNCTION_BLOCK

(* ---- FB_PneumoCollapseControl.st ---- *)
FUNCTION_BLOCK FB_PneumoCollapseControl
VAR_INPUT
	xEnable : BOOL; // Разрешение работы блока (TRUE - автоматический режим)
	xManualStart : BOOL; // Сигнал ручного запуска системы
	tActiveTime : TIME := T#3S; // Время активной работы пневмообрушения
	tPauseCycle : TIME := T#5S; // Время паузы между циклами
	tPauseFB : TIME := T#30S; // Время паузы ФБ между подходами
	nCycleCount : INT := 3; // Количество срабатываний в одном подходе
END_VAR
VAR_OUTPUT
	xPneumoActive : BOOL; // Сигнал управления системой пневмообрушения
	tTimeToNext : TIME; // Время до следующего срабатывания
END_VAR
VAR
	// Внутренние состояния
	eState : E_VibratorState := E_VibratorState.IDLE; // Текущее состояние автоматического цикла
	nCurrentCycle : INT := 0; // Текущий счётчик срабатываний

	// Таймеры
	tonActiveWork : TON; // Таймер активной работы
	tonPauseCycle : TON; // Таймер паузы между циклами
	tonPauseFB : TON; // Таймер паузы ФБ

	// Вспомогательные переменные
	_xManualStartPrev : BOOL; // Предыдущее состояние ручного пуска
	_rtManualStart : R_TRIG; // Детектор фронта ручного пуска
END_VAR

// ========================================
// ДЕТЕКТОР ФРОНТА РУЧНОГО ПУСКА
// ========================================
_rtManualStart(CLK := xManualStart);

// ========================================
// РУЧНОЙ РЕЖИМ УПРАВЛЕНИЯ
// ========================================
IF xManualStart THEN
	// Остановить все таймеры автоматического цикла
	tonActiveWork(IN := FALSE);
	tonPauseCycle(IN := FALSE);
	tonPauseFB(IN := FALSE);

	// Сбросить состояние в IDLE при ручном управлении
	IF NOT _xManualStartPrev THEN
		eState := E_VibratorState.IDLE;
		nCurrentCycle := 0;
	END_IF

	// Ручной запуск системы пневмообрушения
	xPneumoActive := TRUE;

ELSE
	// ========================================
	// АВТОМАТИЧЕСКИЙ РЕЖИМ УПРАВЛЕНИЯ
	// ========================================

	IF NOT xEnable THEN
		// Если Enable выключен - остановить систему и сбросить состояние
		xPneumoActive := FALSE;

		// Сброс состояния
		eState := E_VibratorState.IDLE;
		nCurrentCycle := 0;
		tonActiveWork(IN := FALSE);
		tonPauseCycle(IN := FALSE);
		tonPauseFB(IN := FALSE);

	ELSE
		// Автоматический цикл работы
		CASE eState OF
			E_VibratorState.IDLE:
				// Ожидание старта автоматического цикла
				nCurrentCycle := 0;
				tonActiveWork(IN := FALSE);
				tonPauseCycle(IN := FALSE);
				tonPauseFB(IN := FALSE);
				xPneumoActive := FALSE;

				// Автоматический старт при наличии Enable
				eState := E_VibratorState.ACTIVE_WORK;

			E_VibratorState.ACTIVE_WORK:
				// Активная работа системы пневмообрушения
				tonActiveWork(IN := TRUE, PT := tActiveTime);
				tonPauseCycle(IN := FALSE);
				tonPauseFB(IN := FALSE);

				// Включение системы
				xPneumoActive := TRUE;

				// Переход в паузу после окончания времени активной работы
				IF tonActiveWork.Q THEN
					tonActiveWork(IN := FALSE);
					nCurrentCycle := nCurrentCycle + 1;

					IF nCurrentCycle >= nCycleCount THEN
						// Достигнуто максимальное количество циклов - переход в паузу ФБ
						eState := E_VibratorState.PAUSE_FB;
					ELSE
						// Ещё не достигнуто - переход в паузу между циклами
						eState := E_VibratorState.PAUSE_VIBRATOR;
					END_IF
				END_IF

			E_VibratorState.PAUSE_VIBRATOR:
				// Пауза между циклами
				tonActiveWork(IN := FALSE);
				tonPauseCycle(IN := TRUE, PT := tPauseCycle);
				tonPauseFB(IN := FALSE);

				// Остановка системы
				xPneumoActive := FALSE;

				// Переход обратно в активную работу после паузы
				IF tonPauseCycle.Q THEN
					tonPauseCycle(IN := FALSE);
					eState := E_VibratorState.ACTIVE_WORK;
				END_IF

			E_VibratorState.PAUSE_FB:
				// Пауза между подходами (после достижения nCycleCount)
				tonActiveWork(IN := FALSE);
				tonPauseCycle(IN := FALSE);
				tonPauseFB(IN := TRUE, PT := tPauseFB);

				// Остановка системы
				xPneumoActive := FALSE;

				// Переход в IDLE после паузы и сброс счётчика
				IF tonPauseFB.Q THEN
					tonPauseFB(IN := FALSE);
					nCurrentCycle := 0;
					eState := E_VibratorState.IDLE;
				END_IF
		END_CASE
	END_IF
END_IF

// ========================================
// РАСЧЁТ ВРЕМЕНИ ДО СЛЕДУЮЩЕГО СРАБАТЫВАНИЯ
// ========================================
CASE eState OF
	E_VibratorState.IDLE:
		tTimeToNext := T#0S;

	E_VibratorState.ACTIVE_WORK:
		tTimeToNext := tActiveTime - tonActiveWork.ET;

	E_VibratorState.PAUSE_VIBRATOR:
		tTimeToNext := tPauseCycle - tonPauseCycle.ET;

	E_VibratorState.PAUSE_FB:
		tTimeToNext := tPauseFB - tonPauseFB.ET;
END_CASE

// Сохранение предыдущего состояния ручного пуска
_xManualStartPrev := xManualStart;

END_FUNCTION_BLOCK
